LIN {X -174.485,Y -231.635,Z 231.220,A 53.010,B 90.000,C 0.000} C_DIS
LIN {X -172.527,Y -233.097,Z 231.745,A 53.493,B 90.000,C 0.000} C_DIS
LIN {X -170.564,Y -234.537,Z 232.313,A 53.974,B 90.000,C 0.000} C_DIS
LIN {X -168.598,Y -235.954,Z 232.925,A 54.453,B 90.000,C 0.000} C_DIS
LIN {X -166.629,Y -237.349,Z 233.579,A 54.929,B 90.000,C 0.000} C_DIS
LIN {X -164.658,Y -238.720,Z 234.275,A 55.404,B 90.000,C 0.000} C_DIS
LIN {X -162.687,Y -240.067,Z 235.015,A 55.876,B 90.000,C 0.000} C_DIS
LIN {X -160.716,Y -241.392,Z 235.795,A 56.345,B 90.000,C 0.000} C_DIS
LIN {X -158.746,Y -242.692,Z 236.618,A 56.811,B 90.000,C 0.000} C_DIS
LIN {X -157.556,Y -243.467,Z 237.135,A 57.092,B 90.000,C 0.000} C_DIS
LIN {X -156.469,Y -241.788,Z 237.135,A 57.092,B 90.000,C 0.000} C_DIS
WAIT SEC 0.1
RET=EKI_SetBool("oxy","torchState",FALSE)
RET = EKI_Send("oxy","torchState")
LIN {X -146.690,Y -226.676,Z 237.135,A 57.092,B 90.000,C 0.000} C_DIS
LIN {X -123.076,Y -240.317,Z 224.158,A 62.881,B 90.000,C 0.000} C_DIS
LIN {X -131.281,Y -256.338,Z 224.158,A 62.881,B 90.000,C 0.000} C_DIS
LIN {X -132.192,Y -258.119,Z 224.158,A 62.881,B 90.000,C 0.000} C_DIS
WAIT SEC 1.75
RET=EKI_SetBool("oxy","torchState",TRUE)
RET = EKI_Send("oxy","torchState")
LIN {X -129.997,Y -259.231,Z 224.597,A 63.368,B 90.000,C 0.000} C_DIS
LIN {X -127.784,Y -260.329,Z 224.980,A 63.856,B 90.000,C 0.000} C_DIS
LIN {X -125.556,Y -261.409,Z 225.324,A 64.345,B 90.000,C 0.000} C_DIS
LIN {X -123.317,Y -262.472,Z 225.647,A 64.834,B 90.000,C 0.000} C_DIS
LIN {X -121.069,Y -263.517,Z 225.964,A 65.324,B 90.000,C 0.000} C_DIS
LIN {X -118.813,Y -264.544,Z 226.289,A 65.814,B 90.000,C 0.000} C_DIS
LIN {X -116.551,Y -265.548,Z 226.642,A 66.303,B 90.000,C 0.000} C_DIS
LIN {X -114.287,Y -266.530,Z 227.038,A 66.791,B 90.000,C 0.000} C_DIS
LIN {X -112.023,Y -267.490,Z 227.491,A 67.276,B 90.000,C 0.000} C_DIS
LIN {X -109.763,Y -268.425,Z 228.003,A 67.760,B 90.000,C 0.000} C_DIS
LIN {X -107.506,Y -269.337,Z 228.573,A 68.241,B 90.000,C 0.000} C_DIS
LIN {X -105.255,Y -270.224,Z 229.202,A 68.719,B 90.000,C 0.000} C_DIS
LIN {X -103.012,Y -271.087,Z 229.888,A 69.193,B 90.000,C 0.000} C_DIS
LIN {X -100.777,Y -271.926,Z 230.630,A 69.665,B 90.000,C 0.000} C_DIS
LIN {X -98.553,Y -272.740,Z 231.430,A 70.133,B 90.000,C 0.000} C_DIS
LIN {X -96.341,Y -273.529,Z 232.285,A 70.597,B 90.000,C 0.000} C_DIS
LIN {X -94.142,Y -274.293,Z 233.197,A 71.057,B 90.000,C 0.000} C_DIS
LIN {X -91.959,Y -275.033,Z 234.163,A 71.512,B 90.000,C 0.000} C_DIS
LIN {X -89.792,Y -275.748,Z 235.184,A 71.963,B 90.000,C 0.000} C_DIS
LIN {X -87.644,Y -276.439,Z 236.259,A 72.409,B 90.000,C 0.000} C_DIS
LIN {X -85.515,Y -277.105,Z 237.388,A 72.850,B 90.000,C 0.000} C_DIS
LIN {X -85.176,Y -277.209,Z 237.573,A 72.920,B 90.000,C 0.000} C_DIS
LIN {X -84.588,Y -275.298,Z 237.573,A 72.920,B 90.000,C 0.000} C_DIS
WAIT SEC 0.1
RET=EKI_SetBool("oxy","torchState",FALSE)
RET = EKI_Send("oxy","torchState")
LIN {X -79.302,Y -258.092,Z 237.573,A 72.920,B 90.000,C 0.000} C_DIS
LIN {X -88.721,Y -255.007,Z 203.676,A 70.816,B 90.000,C 0.000} C_DIS
LIN {X -94.636,Y -272.007,Z 203.676,A 70.816,B 90.000,C 0.000} C_DIS
LIN {X -95.293,Y -273.896,Z 203.676,A 70.816,B 90.000,C 0.000} C_DIS
WAIT SEC 1.75
RET=EKI_SetBool("oxy","torchState",TRUE)
RET = EKI_Send("oxy","torchState")
LIN {X -97.616,Y -273.077,Z 203.247,A 70.330,B 90.000,C 0.000} C_DIS
LIN {X -99.938,Y -272.235,Z 202.861,A 69.842,B 90.000,C 0.000} C_DIS
LIN {X -102.254,Y -271.373,Z 202.486,A 69.354,B 90.000,C 0.000} C_DIS
LIN {X -104.561,Y -270.494,Z 202.097,A 68.866,B 90.000,C 0.000} C_DIS
LIN {X -106.853,Y -269.596,Z 201.662,A 68.379,B 90.000,C 0.000} C_DIS
LIN {X -109.130,Y -268.682,Z 201.183,A 67.895,B 90.000,C 0.000} C_DIS
LIN {X -111.390,Y -267.754,Z 200.657,A 67.412,B 90.000,C 0.000} C_DIS
LIN {X -113.632,Y -266.810,Z 200.082,A 66.931,B 90.000,C 0.000} C_DIS
LIN {X -115.856,Y -265.851,Z 199.461,A 66.453,B 90.000,C 0.000} C_DIS
LIN {X -118.061,Y -264.880,Z 198.796,A 65.977,B 90.000,C 0.000} C_DIS
LIN {X -120.246,Y -263.896,Z 198.084,A 65.503,B 90.000,C 0.000} C_DIS
LIN {X -122.409,Y -262.899,Z 197.325,A 65.033,B 90.000,C 0.000} C_DIS
LIN {X -124.550,Y -261.891,Z 196.521,A 64.565,B 90.000,C 0.000} C_DIS
LIN {X -126.670,Y -260.873,Z 195.673,A 64.101,B 90.000,C 0.000} C_DIS
LIN {X -128.766,Y -259.845,Z 194.779,A 63.639,B 90.000,C 0.000} C_DIS
LIN {X -130.837,Y -258.807,Z 193.840,A 63.182,B 90.000,C 0.000} C_DIS
LIN {X -132.884,Y -257.762,Z 192.856,A 62.728,B 90.000,C 0.000} C_DIS
LIN {X -134.776,Y -256.779,Z 191.899,A 62.306,B 90.000,C 0.000} C_DIS
LIN {X -133.846,Y -255.008,Z 191.899,A 62.306,B 90.000,C 0.000} C_DIS
WAIT SEC 0.1
RET=EKI_SetBool("oxy","torchState",FALSE)
RET = EKI_Send("oxy","torchState")
LIN {X -125.481,Y -239.070,Z 191.899,A 62.306,B 90.000,C 0.000} C_DIS
LIN {X -100.690,Y -250.523,Z 169.381,A 68.104,B 90.000,C 0.000} C_DIS
LIN {X -107.403,Y -267.224,Z 169.381,A 68.104,B 90.000,C 0.000} C_DIS
LIN {X -108.148,Y -269.080,Z 169.381,A 68.104,B 90.000,C 0.000} C_DIS
WAIT SEC 1.75
RET=EKI_SetBool("oxy","torchState",TRUE)
RET = EKI_Send("oxy","torchState")
LIN {X -105.841,Y -269.995,Z 169.670,A 68.594,B 90.000,C 0.000} C_DIS
LIN {X -103.520,Y -270.893,Z 169.913,A 69.086,B 90.000,C 0.000} C_DIS
LIN {X -101.192,Y -271.772,Z 170.145,A 69.578,B 90.000,C 0.000} C_DIS
LIN {X -98.858,Y -272.630,Z 170.404,A 70.069,B 90.000,C 0.000} C_DIS
LIN {X -96.524,Y -273.464,Z 170.725,A 70.559,B 90.000,C 0.000} C_DIS
LIN {X -94.192,Y -274.276,Z 171.117,A 71.046,B 90.000,C 0.000} C_DIS
LIN {X -91.865,Y -275.065,Z 171.577,A 71.532,B 90.000,C 0.000} C_DIS
LIN {X -89.544,Y -275.829,Z 172.102,A 72.015,B 90.000,C 0.000} C_DIS
LIN {X -87.230,Y -276.569,Z 172.690,A 72.495,B 90.000,C 0.000} C_DIS
LIN {X -84.924,Y -277.286,Z 173.335,A 72.972,B 90.000,C 0.000} C_DIS
LIN {X -82.626,Y -277.979,Z 174.034,A 73.446,B 90.000,C 0.000} C_DIS
LIN {X -80.337,Y -278.649,Z 174.783,A 73.917,B 90.000,C 0.000} C_DIS
LIN {X -78.058,Y -279.297,Z 175.578,A 74.385,B 90.000,C 0.000} C_DIS
LIN {X -75.788,Y -279.921,Z 176.419,A 74.851,B 90.000,C 0.000} C_DIS
LIN {X -73.526,Y -280.523,Z 177.298,A 75.313,B 90.000,C 0.000} C_DIS
LIN {X -71.273,Y -281.105,Z 178.212,A 75.773,B 90.000,C 0.000} C_DIS
LIN {X -69.029,Y -281.664,Z 179.160,A 76.230,B 90.000,C 0.000} C_DIS
LIN {X -66.792,Y -282.203,Z 180.136,A 76.684,B 90.000,C 0.000} C_DIS
LIN {X -64.561,Y -282.722,Z 181.137,A 77.137,B 90.000,C 0.000} C_DIS
LIN {X -62.337,Y -283.220,Z 182.163,A 77.587,B 90.000,C 0.000} C_DIS
LIN {X -60.117,Y -283.699,Z 183.208,A 78.036,B 90.000,C 0.000} C_DIS
LIN {X -57.901,Y -284.159,Z 184.270,A 78.483,B 90.000,C 0.000} C_DIS
LIN {X -55.688,Y -284.600,Z 185.345,A 78.929,B 90.000,C 0.000} C_DIS
LIN {X -53.477,Y -285.024,Z 186.431,A 79.374,B 90.000,C 0.000} C_DIS
LIN {X -51.266,Y -285.431,Z 187.524,A 79.818,B 90.000,C 0.000} C_DIS
LIN {X -49.054,Y -285.816,Z 188.623,A 80.261,B 90.000,C 0.000} C_DIS
LIN {X -47.559,Y -286.074,Z 189.367,A 80.561,B 90.000,C 0.000} C_DIS
LIN {X -47.231,Y -284.101,Z 189.367,A 80.561,B 90.000,C 0.000} C_DIS
WAIT SEC 0.1
RET=EKI_SetBool("oxy","torchState",FALSE)
RET = EKI_Send("oxy","torchState")
LIN {X -44.279,Y -266.344,Z 189.367,A 80.561,B 90.000,C 0.000} C_DIS
LIN {X -23.730,Y -268.955,Z 178.464,A 84.958,B 90.000,C 0.000} C_DIS
LIN {X -25.312,Y -286.885,Z 178.464,A 84.958,B 90.000,C 0.000} C_DIS
LIN {X -25.488,Y -288.878,Z 178.464,A 84.958,B 90.000,C 0.000} C_DIS
WAIT SEC 1.75
RET=EKI_SetBool("oxy","torchState",TRUE)
RET = EKI_Send("oxy","torchState")
LIN {X -27.825,Y -288.662,Z 177.602,A 84.494,B 90.000,C 0.000} C_DIS
LIN {X -30.135,Y -288.429,Z 176.676,A 84.035,B 90.000,C 0.000} C_DIS
LIN {X -32.420,Y -288.182,Z 175.693,A 83.581,B 90.000,C 0.000} C_DIS
LIN {X -34.681,Y -287.919,Z 174.660,A 83.132,B 90.000,C 0.000} C_DIS
LIN {X -36.919,Y -287.640,Z 173.581,A 82.686,B 90.000,C 0.000} C_DIS
LIN {X -39.139,Y -287.347,Z 172.471,A 82.244,B 90.000,C 0.000} C_DIS
LIN {X -41.342,Y -287.038,Z 171.331,A 81.804,B 90.000,C 0.000} C_DIS
LIN {X -43.532,Y -286.713,Z 170.171,A 81.367,B 90.000,C 0.000} C_DIS
LIN {X -45.713,Y -286.374,Z 168.998,A 80.931,B 90.000,C 0.000} C_DIS
LIN {X -47.888,Y -286.018,Z 167.817,A 80.495,B 90.000,C 0.000} C_DIS
LIN {X -50.060,Y -285.644,Z 166.638,A 80.060,B 90.000,C 0.000} C_DIS
LIN {X -52.233,Y -285.256,Z 165.466,A 79.624,B 90.000,C 0.000} C_DIS
LIN {X -54.410,Y -284.849,Z 164.306,A 79.186,B 90.000,C 0.000} C_DIS
LIN {X -56.595,Y -284.423,Z 163.169,A 78.746,B 90.000,C 0.000} C_DIS
LIN {X -58.790,Y -283.978,Z 162.059,A 78.304,B 90.000,C 0.000} C_DIS
LIN {X -60.381,Y -283.644,Z 161.280,A 77.983,B 90.000,C 0.000} C_DIS
LIN {X -59.964,Y -281.688,Z 161.280,A 77.983,B 90.000,C 0.000} C_DIS
WAIT SEC 0.1
RET=EKI_SetBool("oxy","torchState",FALSE)
RET = EKI_Send("oxy","torchState")
LIN {X -56.216,Y -264.083,Z 161.280,A 77.983,B 90.000,C 0.000} C_DIS
LIN {X -40.841,Y -266.893,Z 146.065,A 81.300,B 90.000,C 0.000} C_DIS
LIN {X -43.563,Y -284.686,Z 146.065,A 81.300,B 90.000,C 0.000} C_DIS
LIN {X -43.866,Y -286.663,Z 146.065,A 81.300,B 90.000,C 0.000} C_DIS
WAIT SEC 1.75
RET=EKI_SetBool("oxy","torchState",TRUE)
RET = EKI_Send("oxy","torchState")
LIN {X -41.493,Y -287.012,Z 146.771,A 81.774,B 90.000,C 0.000} C_DIS
LIN {X -39.121,Y -287.344,Z 147.484,A 82.247,B 90.000,C 0.000} C_DIS
LIN {X -36.747,Y -287.661,Z 148.202,A 82.720,B 90.000,C 0.000} C_DIS
LIN {X -34.373,Y -287.952,Z 148.929,A 83.193,B 90.000,C 0.000} C_DIS
LIN {X -32.000,Y -288.224,Z 149.663,A 83.665,B 90.000,C 0.000} C_DIS
LIN {X -29.626,Y -288.481,Z 150.403,A 84.137,B 90.000,C 0.000} C_DIS
LIN {X -27.252,Y -288.713,Z 151.151,A 84.608,B 90.000,C 0.000} C_DIS
LIN {X -24.879,Y -288.926,Z 151.907,A 85.079,B 90.000,C 0.000} C_DIS
LIN {X -22.506,Y -289.123,Z 152.668,A 85.549,B 90.000,C 0.000} C_DIS
LIN {X -20.134,Y -289.297,Z 153.437,A 86.019,B 90.000,C 0.000} C_DIS
LIN {X -18.908,Y -289.383,Z 153.837,A 86.262,B 90.000,C 0.000} C_DIS
LIN {X -18.777,Y -287.387,Z 153.837,A 86.262,B 90.000,C 0.000} C_DIS
WAIT SEC 0.1
RET=EKI_SetBool("oxy","torchState",FALSE)
RET = EKI_Send("oxy","torchState")
LIN {X -17.604,Y -269.426,Z 153.837,A 86.262,B 90.000,C 0.000} C_DIS
LIN {X 5.612,Y -269.942,Z 139.862,A 91.191,B 90.000,C 0.000} C_DIS
LIN {X 5.986,Y -287.938,Z 139.862,A 91.191,B 90.000,C 0.000} C_DIS
LIN {X 6.028,Y -289.937,Z 139.862,A 91.191,B 90.000,C 0.000} C_DIS
WAIT SEC 1.75
RET=EKI_SetBool("oxy","torchState",TRUE)
RET = EKI_Send("oxy","torchState")
LIN {X 8.397,Y -289.878,Z 140.657,A 91.659,B 90.000,C 0.000} C_DIS
LIN {X 10.728,Y -289.801,Z 141.555,A 92.120,B 90.000,C 0.000} C_DIS
LIN {X 13.001,Y -289.708,Z 142.592,A 92.569,B 90.000,C 0.000} C_DIS
LIN {X 15.183,Y -289.602,Z 143.807,A 93.001,B 90.000,C 0.000} C_DIS
LIN {X 17.238,Y -289.487,Z 145.226,A 93.408,B 90.000,C 0.000} C_DIS
LIN {X 19.120,Y -289.369,Z 146.866,A 93.780,B 90.000,C 0.000} C_DIS
LIN {X 20.776,Y -289.255,Z 148.735,A 94.108,B 90.000,C 0.000} C_DIS
LIN {X 22.142,Y -289.153,Z 150.827,A 94.379,B 90.000,C 0.000} C_DIS
LIN {X 22.275,Y -289.143,Z 151.073,A 94.405,B 90.000,C 0.000} C_DIS
LIN {X 22.122,Y -287.149,Z 151.073,A 94.405,B 90.000,C 0.000} C_DIS
WAIT SEC 0.1
RET=EKI_SetBool("oxy","torchState",FALSE)
RET = EKI_Send("oxy","torchState")
LIN {X 20.739,Y -269.202,Z 151.073,A 94.405,B 90.000,C 0.000} C_DIS
LIN {X 20.977,Y -269.184,Z 165.846,A 94.456,B 90.000,C 0.000} C_DIS
LIN {X 22.376,Y -287.129,Z 165.846,A 94.456,B 90.000,C 0.000} C_DIS
LIN {X 22.531,Y -289.123,Z 165.846,A 94.456,B 90.000,C 0.000} C_DIS
WAIT SEC 1.75
RET=EKI_SetBool("oxy","torchState",TRUE)
RET = EKI_Send("oxy","torchState")
LIN {X 21.416,Y -289.208,Z 168.082,A 94.235,B 90.000,C 0.000} C_DIS
LIN {X 20.047,Y -289.306,Z 170.171,A 93.964,B 90.000,C 0.000} C_DIS
LIN {X 18.459,Y -289.412,Z 172.099,A 93.649,B 90.000,C 0.000} C_DIS
LIN {X 16.685,Y -289.520,Z 173.857,A 93.298,B 90.000,C 0.000} C_DIS
LIN {X 14.754,Y -289.624,Z 175.441,A 92.916,B 90.000,C 0.000} C_DIS
LIN {X 12.689,Y -289.722,Z 176.845,A 92.508,B 90.000,C 0.000} C_DIS
LIN {X 10.513,Y -289.809,Z 178.073,A 92.078,B 90.000,C 0.000} C_DIS
LIN {X 8.247,Y -289.883,Z 179.127,A 91.630,B 90.000,C 0.000} C_DIS
LIN {X 5.908,Y -289.940,Z 180.005,A 91.167,B 90.000,C 0.000} C_DIS
LIN {X 3.512,Y -289.979,Z 180.716,A 90.694,B 90.000,C 0.000} C_DIS
LIN {X 1.073,Y -289.998,Z 181.264,A 90.212,B 90.000,C 0.000} C_DIS
LIN {X -1.396,Y -289.997,Z 181.653,A 89.724,B 90.000,C 0.000} C_DIS
LIN {X -3.885,Y -289.974,Z 181.888,A 89.232,B 90.000,C 0.000} C_DIS
LIN {X -6.286,Y -289.932,Z 181.974,A 88.758,B 90.000,C 0.000} C_DIS
LIN {X -6.243,Y -287.932,Z 181.974,A 88.758,B 90.000,C 0.000} C_DIS
WAIT SEC 0.1
RET=EKI_SetBool("oxy","torchState",FALSE)
RET = EKI_Send("oxy","torchState")
LIN {X -5.852,Y -269.937,Z 181.974,A 88.758,B 90.000,C 0.000} C_DIS
LIN {X -12.189,Y -269.725,Z 203.494,A 87.412,B 90.000,C 0.000} C_DIS
LIN {X -13.002,Y -287.706,Z 203.494,A 87.412,B 90.000,C 0.000} C_DIS
LIN {X -13.092,Y -289.704,Z 203.494,A 87.412,B 90.000,C 0.000} C_DIS
WAIT SEC 1.75
RET=EKI_SetBool("oxy","torchState",TRUE)
RET = EKI_Send("oxy","torchState")
LIN {X -10.663,Y -289.804,Z 204.075,A 87.893,B 90.000,C 0.000} C_DIS
LIN {X -8.217,Y -289.883,Z 204.584,A 88.376,B 90.000,C 0.000} C_DIS
LIN {X -5.755,Y -289.942,Z 205.016,A 88.863,B 90.000,C 0.000} C_DIS
LIN {X -3.281,Y -289.981,Z 205.369,A 89.352,B 90.000,C 0.000} C_DIS
LIN {X -0.796,Y -289.999,Z 205.637,A 89.843,B 90.000,C 0.000} C_DIS
LIN {X 1.698,Y -289.995,Z 205.815,A 90.335,B 90.000,C 0.000} C_DIS
LIN {X 4.196,Y -289.970,Z 205.903,A 90.829,B 90.000,C 0.000} C_DIS
LIN {X 6.695,Y -289.922,Z 205.890,A 91.323,B 90.000,C 0.000} C_DIS
LIN {X 9.191,Y -289.854,Z 205.779,A 91.816,B 90.000,C 0.000} C_DIS
LIN {X 11.679,Y -289.764,Z 205.556,A 92.308,B 90.000,C 0.000} C_DIS
LIN {X 14.154,Y -289.654,Z 205.224,A 92.798,B 90.000,C 0.000} C_DIS
LIN {X 16.610,Y -289.524,Z 204.776,A 93.283,B 90.000,C 0.000} C_DIS
LIN {X 19.039,Y -289.374,Z 204.206,A 93.764,B 90.000,C 0.000} C_DIS
LIN {X 21.435,Y -289.206,Z 203.512,A 94.239,B 90.000,C 0.000} C_DIS
LIN {X 23.790,Y -289.023,Z 202.694,A 94.705,B 90.000,C 0.000} C_DIS
LIN {X 23.626,Y -287.029,Z 202.694,A 94.705,B 90.000,C 0.000} C_DIS
WAIT SEC 0.1
RET=EKI_SetBool("oxy","torchState",FALSE)
RET = EKI_Send("oxy","torchState")
LIN {X 22.149,Y -269.090,Z 202.694,A 94.705,B 90.000,C 0.000} C_DIS
LIN {X 39.945,Y -267.029,Z 190.477,A 98.508,B 90.000,C 0.000} C_DIS
LIN {X 42.608,Y -284.831,Z 190.477,A 98.508,B 90.000,C 0.000} C_DIS
LIN {X 42.904,Y -286.809,Z 190.477,A 98.508,B 90.000,C 0.000} C_DIS
WAIT SEC 1.75
RET=EKI_SetBool("oxy","torchState",TRUE)
RET = EKI_Send("oxy","torchState")
LIN {X 44.729,Y -286.530,Z 188.792,A 98.873,B 90.000,C 0.000} C_DIS
LIN {X 46.502,Y -286.247,Z 187.053,A 99.227,B 90.000,C 0.000} C_DIS
LIN {X 48.216,Y -285.963,Z 185.256,A 99.571,B 90.000,C 0.000} C_DIS
LIN {X 49.864,Y -285.681,Z 183.398,A 99.901,B 90.000,C 0.000} C_DIS
LIN {X 51.432,Y -285.403,Z 181.471,A 100.216,B 90.000,C 0.000} C_DIS
LIN {X 52.915,Y -285.131,Z 179.477,A 100.513,B 90.000,C 0.000} C_DIS
LIN {X 54.300,Y -284.871,Z 177.412,A 100.792,B 90.000,C 0.000} C_DIS
LIN {X 55.573,Y -284.625,Z 175.275,A 101.048,B 90.000,C 0.000} C_DIS
LIN {X 56.724,Y -284.398,Z 173.068,A 101.280,B 90.000,C 0.000} C_DIS
LIN {X 57.368,Y -284.269,Z 171.672,A 101.410,B 90.000,C 0.000} C_DIS
LIN {X 56.973,Y -282.309,Z 171.672,A 101.410,B 90.000,C 0.000} C_DIS
WAIT SEC 0.1
RET=EKI_SetBool("oxy","torchState",FALSE)
RET = EKI_Send("oxy","torchState")
LIN {X 53.412,Y -264.664,Z 171.672,A 101.410,B 90.000,C 0.000} C_DIS
LIN {X 54.636,Y -264.414,Z 148.285,A 101.675,B 90.000,C 0.000} C_DIS
LIN {X 58.279,Y -282.042,Z 148.285,A 101.675,B 90.000,C 0.000} C_DIS
LIN {X 58.684,Y -284.000,Z 148.285,A 101.675,B 90.000,C 0.000} C_DIS
WAIT SEC 1.75
RET=EKI_SetBool("oxy","torchState",TRUE)
RET = EKI_Send("oxy","torchState")
LIN {X 57.692,Y -284.204,Z 146.000,A 101.475,B 90.000,C 0.000} C_DIS
LIN {X 56.490,Y -284.445,Z 143.821,A 101.233,B 90.000,C 0.000} C_DIS
LIN {X 55.104,Y -284.717,Z 141.759,A 100.954,B 90.000,C 0.000} C_DIS
LIN {X 53.557,Y -285.012,Z 139.817,A 100.642,B 90.000,C 0.000} C_DIS
LIN {X 51.869,Y -285.324,Z 138.000,A 100.303,B 90.000,C 0.000} C_DIS
LIN {X 50.060,Y -285.646,Z 136.306,A 99.940,B 90.000,C 0.000} C_DIS
LIN {X 48.146,Y -285.975,Z 134.731,A 99.557,B 90.000,C 0.000} C_DIS
LIN {X 47.860,Y -286.023,Z 134.510,A 99.499,B 90.000,C 0.000} C_DIS
LIN {X 47.530,Y -284.051,Z 134.510,A 99.499,B 90.000,C 0.000} C_DIS
WAIT SEC 0.1
RET=EKI_SetBool("oxy","torchState",FALSE)
RET = EKI_Send("oxy","torchState")
LIN {X 44.559,Y -266.298,Z 134.510,A 99.499,B 90.000,C 0.000} C_DIS
LIN {X 30.080,Y -268.319,Z 126.079,A 96.396,B 90.000,C 0.000} C_DIS
LIN {X 32.085,Y -286.207,Z 126.079,A 96.396,B 90.000,C 0.000} C_DIS
LIN {X 32.308,Y -288.195,Z 126.079,A 96.396,B 90.000,C 0.000} C_DIS
WAIT SEC 1.75
RET=EKI_SetBool("oxy","torchState",TRUE)
RET = EKI_Send("oxy","torchState")
LIN {X 30.008,Y -288.442,Z 125.131,A 95.939,B 90.000,C 0.000} C_DIS
LIN {X 27.696,Y -288.674,Z 124.211,A 95.480,B 90.000,C 0.000} C_DIS
LIN {X 25.369,Y -288.887,Z 123.323,A 95.019,B 90.000,C 0.000} C_DIS
LIN {X 23.028,Y -289.083,Z 122.466,A 94.555,B 90.000,C 0.000} C_DIS
LIN {X 20.675,Y -289.261,Z 121.643,A 94.088,B 90.000,C 0.000} C_DIS
LIN {X 18.308,Y -289.421,Z 120.853,A 93.620,B 90.000,C 0.000} C_DIS
LIN {X 15.929,Y -289.561,Z 120.099,A 93.149,B 90.000,C 0.000} C_DIS
LIN {X 13.538,Y -289.683,Z 119.381,A 92.676,B 90.000,C 0.000} C_DIS
LIN {X 11.135,Y -289.785,Z 118.702,A 92.200,B 90.000,C 0.000} C_DIS
LIN {X 8.720,Y -289.869,Z 118.059,A 91.723,B 90.000,C 0.000} C_DIS
LIN {X 6.295,Y -289.931,Z 117.459,A 91.244,B 90.000,C 0.000} C_DIS
LIN {X 3.859,Y -289.974,Z 116.898,A 90.762,B 90.000,C 0.000} C_DIS
LIN {X 1.414,Y -289.996,Z 116.380,A 90.279,B 90.000,C 0.000} C_DIS
LIN {X -1.041,Y -289.997,Z 115.907,A 89.794,B 90.000,C 0.000} C_DIS
LIN {X -3.503,Y -289.978,Z 115.477,A 89.308,B 90.000,C 0.000} C_DIS
LIN {X -5.973,Y -289.938,Z 115.094,A 88.820,B 90.000,C 0.000} C_DIS
LIN {X -8.450,Y -289.876,Z 114.760,A 88.330,B 90.000,C 0.000} C_DIS
LIN {X -10.931,Y -289.793,Z 114.474,A 87.840,B 90.000,C 0.000} C_DIS
LIN {X -13.418,Y -289.689,Z 114.237,A 87.348,B 90.000,C 0.000} C_DIS
LIN {X -15.907,Y -289.563,Z 114.051,A 86.856,B 90.000,C 0.000} C_DIS
LIN {X -18.399,Y -289.415,Z 113.920,A 86.362,B 90.000,C 0.000} C_DIS
LIN {X -20.892,Y -289.246,Z 113.843,A 85.869,B 90.000,C 0.000} C_DIS
LIN {X -23.384,Y -289.055,Z 113.821,A 85.375,B 90.000,C 0.000} C_DIS
LIN {X -25.875,Y -288.843,Z 113.854,A 84.881,B 90.000,C 0.000} C_DIS
LIN {X -26.365,Y -288.799,Z 113.866,A 84.784,B 90.000,C 0.000} C_DIS
LIN {X -26.184,Y -286.807,Z 113.866,A 84.784,B 90.000,C 0.000} C_DIS
WAIT SEC 0.1
RET=EKI_SetBool("oxy","torchState",FALSE)
RET = EKI_Send("oxy","torchState")
LIN {X -24.547,Y -268.882,Z 113.866,A 84.784,B 90.000,C 0.000} C_DIS
LIN {X -36.877,Y -267.470,Z 113.990,A 82.150,B 90.000,C 0.000} C_DIS
LIN {X -39.336,Y -285.301,Z 113.990,A 82.150,B 90.000,C 0.000} C_DIS
LIN {X -39.609,Y -287.282,Z 113.990,A 82.150,B 90.000,C 0.000} C_DIS
WAIT SEC 1.75
RET=EKI_SetBool("oxy","torchState",TRUE)
RET = EKI_Send("oxy","torchState")
LIN {X -42.062,Y -286.933,Z 113.662,A 81.660,B 90.000,C 0.000} C_DIS
LIN {X -44.477,Y -286.569,Z 113.127,A 81.178,B 90.000,C 0.000} C_DIS
LIN {X -46.822,Y -286.195,Z 112.348,A 80.709,B 90.000,C 0.000} C_DIS
LIN {X -49.059,Y -285.820,Z 111.296,A 80.261,B 90.000,C 0.000} C_DIS
LIN {X -51.128,Y -285.457,Z 109.942,A 79.845,B 90.000,C 0.000} C_DIS
LIN {X -52.966,Y -285.122,Z 108.282,A 79.476,B 90.000,C 0.000} C_DIS
LIN {X -54.526,Y -284.828,Z 106.351,A 79.163,B 90.000,C 0.000} C_DIS
LIN {X -55.790,Y -284.583,Z 104.208,A 78.908,B 90.000,C 0.000} C_DIS
LIN {X -56.744,Y -284.394,Z 101.905,A 78.716,B 90.000,C 0.000} C_DIS
LIN {X -57.169,Y -284.309,Z 100.461,A 78.631,B 90.000,C 0.000} C_DIS
LIN {X -56.774,Y -282.348,Z 100.461,A 78.631,B 90.000,C 0.000} C_DIS
WAIT SEC 0.1
RET=EKI_SetBool("oxy","torchState",FALSE)
RET = EKI_Send("oxy","torchState")
LIN {X -53.226,Y -264.702,Z 100.461,A 78.631,B 90.000,C 0.000} C_DIS
LIN {X -60.163,Y -263.212,Z 120.264,A 77.125,B 90.000,C 0.000} C_DIS
LIN {X -64.173,Y -280.759,Z 120.264,A 77.125,B 90.000,C 0.000} C_DIS
LIN {X -64.619,Y -282.709,Z 120.264,A 77.125,B 90.000,C 0.000} C_DIS
WAIT SEC 1.75
RET=EKI_SetBool("oxy","torchState",TRUE)
RET = EKI_Send("oxy","torchState")
LIN {X -62.571,Y -283.169,Z 121.622,A 77.540,B 90.000,C 0.000} C_DIS
LIN {X -60.462,Y -283.627,Z 122.883,A 77.966,B 90.000,C 0.000} C_DIS
LIN {X -58.301,Y -284.079,Z 124.056,A 78.402,B 90.000,C 0.000} C_DIS
LIN {X -56.093,Y -284.523,Z 125.139,A 78.847,B 90.000,C 0.000} C_DIS
LIN {X -53.844,Y -284.957,Z 126.141,A 79.300,B 90.000,C 0.000} C_DIS
LIN {X -51.560,Y -285.380,Z 127.064,A 79.759,B 90.000,C 0.000} C_DIS
LIN {X -49.244,Y -285.788,Z 127.912,A 80.223,B 90.000,C 0.000} C_DIS
LIN {X -46.902,Y -286.182,Z 128.691,A 80.693,B 90.000,C 0.000} C_DIS
LIN {X -44.537,Y -286.559,Z 129.408,A 81.166,B 90.000,C 0.000} C_DIS
LIN {X -42.359,Y -286.890,Z 130.012,A 81.601,B 90.000,C 0.000} C_DIS
LIN {X -42.067,Y -284.911,Z 130.012,A 81.601,B 90.000,C 0.000} C_DIS
WAIT SEC 0.1
RET=EKI_SetBool("oxy","torchState",FALSE)
RET = EKI_Send("oxy","torchState")
LIN {X -39.438,Y -267.104,Z 130.012,A 81.601,B 90.000,C 0.000} C_DIS
LIN {X -74.388,Y -259.551,Z 101.612,A 74.008,B 90.000,C 0.000} C_DIS
LIN {X -79.347,Y -276.854,Z 101.612,A 74.008,B 90.000,C 0.000} C_DIS
LIN {X -79.898,Y -278.777,Z 101.612,A 74.008,B 90.000,C 0.000} C_DIS
WAIT SEC 1.75
RET=EKI_SetBool("oxy","torchState",TRUE)
RET = EKI_Send("oxy","torchState")
LIN {X -80.728,Y -278.537,Z 99.266,A 73.837,B 90.000,C 0.000} C_DIS
LIN {X -81.396,Y -278.343,Z 96.865,A 73.699,B 90.000,C 0.000} C_DIS
LIN {X -81.903,Y -278.194,Z 94.422,A 73.595,B 90.000,C 0.000} C_DIS
LIN {X -82.243,Y -278.094,Z 91.947,A 73.525,B 90.000,C 0.000} C_DIS
LIN {X -82.420,Y -278.041,Z 89.454,A 73.488,B 90.000,C 0.000} C_DIS
LIN {X -82.435,Y -278.037,Z 86.955,A 73.485,B 90.000,C 0.000} C_DIS
LIN {X -82.285,Y -278.081,Z 84.460,A 73.516,B 90.000,C 0.000} C_DIS
LIN {X -81.969,Y -278.175,Z 81.982,A 73.582,B 90.000,C 0.000} C_DIS
LIN {X -81.493,Y -278.314,Z 79.532,A 73.679,B 90.000,C 0.000} C_DIS
LIN {X -80.862,Y -278.498,Z 77.120,A 73.809,B 90.000,C 0.000} C_DIS
LIN {X -80.077,Y -278.725,Z 74.758,A 73.971,B 90.000,C 0.000} C_DIS
LIN {X -79.144,Y -278.991,Z 72.454,A 74.162,B 90.000,C 0.000} C_DIS
LIN {X -78.069,Y -279.294,Z 70.218,A 74.383,B 90.000,C 0.000} C_DIS
LIN {X -76.855,Y -279.631,Z 68.059,A 74.632,B 90.000,C 0.000} C_DIS
LIN {X -76.252,Y -279.796,Z 67.095,A 74.755,B 90.000,C 0.000} C_DIS
LIN {X -75.726,Y -277.866,Z 67.095,A 74.755,B 90.000,C 0.000} C_DIS
WAIT SEC 0.1
RET=EKI_SetBool("oxy","torchState",FALSE)
RET = EKI_Send("oxy","torchState")
LIN {X -70.994,Y -260.499,Z 67.095,A 74.755,B 90.000,C 0.000} C_DIS
LIN {X -71.477,Y -260.367,Z 43.916,A 74.649,B 90.000,C 0.000} C_DIS
LIN {X -76.242,Y -277.725,Z 43.916,A 74.649,B 90.000,C 0.000} C_DIS
LIN {X -76.772,Y -279.654,Z 43.916,A 74.649,B 90.000,C 0.000} C_DIS
WAIT SEC 1.75
RET=EKI_SetBool("oxy","torchState",TRUE)
RET = EKI_Send("oxy","torchState")
LIN {X -79.027,Y -279.023,Z 44.789,A 74.186,B 90.000,C 0.000} C_DIS
LIN {X -81.275,Y -278.378,Z 45.673,A 73.724,B 90.000,C 0.000} C_DIS
LIN {X -83.506,Y -277.717,Z 46.585,A 73.265,B 90.000,C 0.000} C_DIS
LIN {X -85.712,Y -277.044,Z 47.550,A 72.809,B 90.000,C 0.000} C_DIS
LIN {X -87.883,Y -276.363,Z 48.585,A 72.359,B 90.000,C 0.000} C_DIS
LIN {X -90.009,Y -275.678,Z 49.708,A 71.918,B 90.000,C 0.000} C_DIS
LIN {X -92.072,Y -274.996,Z 50.943,A 71.489,B 90.000,C 0.000} C_DIS
LIN {X -94.061,Y -274.322,Z 52.298,A 71.074,B 90.000,C 0.000} C_DIS
LIN {X -95.956,Y -273.665,Z 53.791,A 70.678,B 90.000,C 0.000} C_DIS
LIN {X -97.736,Y -273.034,Z 55.428,A 70.304,B 90.000,C 0.000} C_DIS
LIN {X -99.376,Y -272.441,Z 57.219,A 69.960,B 90.000,C 0.000} C_DIS
LIN {X -100.671,Y -271.966,Z 58.905,A 69.687,B 90.000,C 0.000} C_DIS
LIN {X -99.977,Y -270.090,Z 58.905,A 69.687,B 90.000,C 0.000} C_DIS
WAIT SEC 0.1
RET=EKI_SetBool("oxy","torchState",FALSE)
RET = EKI_Send("oxy","torchState")
LIN {X -93.728,Y -253.209,Z 58.905,A 69.687,B 90.000,C 0.000} C_DIS
LIN {X -111.983,Y -245.682,Z 45.730,A 65.496,B 90.000,C 0.000} C_DIS
LIN {X -119.449,Y -262.061,Z 45.730,A 65.496,B 90.000,C 0.000} C_DIS
LIN {X -120.278,Y -263.881,Z 45.730,A 65.496,B 90.000,C 0.000} C_DIS
WAIT SEC 1.75
RET=EKI_SetBool("oxy","torchState",TRUE)
RET = EKI_Send("oxy","torchState")
LIN {X -122.345,Y -262.927,Z 46.762,A 65.046,B 90.000,C 0.000} C_DIS
LIN {X -124.405,Y -261.960,Z 47.797,A 64.597,B 90.000,C 0.000} C_DIS
LIN {X -126.462,Y -260.973,Z 48.818,A 64.146,B 90.000,C 0.000} C_DIS
LIN {X -128.524,Y -259.964,Z 49.808,A 63.693,B 90.000,C 0.000} C_DIS
LIN {X -130.597,Y -258.929,Z 50.746,A 63.235,B 90.000,C 0.000} C_DIS
LIN {X -132.685,Y -257.865,Z 51.615,A 62.772,B 90.000,C 0.000} C_DIS
LIN {X -134.794,Y -256.769,Z 52.391,A 62.302,B 90.000,C 0.000} C_DIS
LIN {X -136.923,Y -255.640,Z 53.055,A 61.826,B 90.000,C 0.000} C_DIS
LIN {X -139.071,Y -254.478,Z 53.585,A 61.344,B 90.000,C 0.000} C_DIS
LIN {X -139.508,Y -254.239,Z 53.676,A 61.245,B 90.000,C 0.000} C_DIS
LIN {X -138.546,Y -252.486,Z 53.676,A 61.245,B 90.000,C 0.000} C_DIS
WAIT SEC 0.1
RET=EKI_SetBool("oxy","torchState",FALSE)
RET = EKI_Send("oxy","torchState")
LIN {X -129.886,Y -236.706,Z 53.676,A 61.245,B 90.000,C 0.000} C_DIS
LIN {X -145.274,Y -227.586,Z 52.101,A 57.449,B 90.000,C 0.000} C_DIS
LIN {X -154.959,Y -242.758,Z 52.101,A 57.449,B 90.000,C 0.000} C_DIS
LIN {X -156.035,Y -244.444,Z 52.101,A 57.449,B 90.000,C 0.000} C_DIS
WAIT SEC 1.75
RET=EKI_SetBool("oxy","torchState",TRUE)
RET = EKI_Send("oxy","torchState")
LIN {X -157.996,Y -243.181,Z 51.202,A 56.988,B 90.000,C 0.000} C_DIS
LIN {X -159.895,Y -241.937,Z 50.155,A 56.540,B 90.000,C 0.000} C_DIS
LIN {X -161.724,Y -240.719,Z 48.964,A 56.105,B 90.000,C 0.000} C_DIS
LIN {X -163.476,Y -239.532,Z 47.634,A 55.687,B 90.000,C 0.000} C_DIS
LIN {X -165.147,Y -238.383,Z 46.171,A 55.287,B 90.000,C 0.000} C_DIS
LIN {X -166.728,Y -237.280,Z 44.580,A 54.906,B 90.000,C 0.000} C_DIS
LIN {X -168.215,Y -236.228,Z 42.868,A 54.546,B 90.000,C 0.000} C_DIS
LIN {X -169.324,Y -235.434,Z 41.430,A 54.276,B 90.000,C 0.000} C_DIS
LIN {X -168.157,Y -233.810,Z 41.430,A 54.276,B 90.000,C 0.000} C_DIS
WAIT SEC 0.1
RET=EKI_SetBool("oxy","torchState",FALSE)
RET = EKI_Send("oxy","torchState")
LIN {X -157.647,Y -219.197,Z 41.430,A 54.276,B 90.000,C 0.000} C_DIS
LIN {X -172.149,Y -208.002,Z 56.028,A 50.388,B 90.000,C 0.000} C_DIS
LIN {X -183.626,Y -221.868,Z 56.028,A 50.388,B 90.000,C 0.000} C_DIS
LIN {X -184.901,Y -223.409,Z 56.028,A 50.388,B 90.000,C 0.000} C_DIS
WAIT SEC 1.75
RET=EKI_SetBool("oxy","torchState",TRUE)
RET = EKI_Send("oxy","torchState")
LIN {X -183.131,Y -224.861,Z 57.032,A 50.840,B 90.000,C 0.000} C_DIS
LIN {X -181.357,Y -226.294,Z 58.055,A 51.291,B 90.000,C 0.000} C_DIS
LIN {X -179.578,Y -227.708,Z 59.096,A 51.740,B 90.000,C 0.000} C_DIS
LIN {X -177.795,Y -229.103,Z 60.156,A 52.187,B 90.000,C 0.000} C_DIS
LIN {X -176.008,Y -230.479,Z 61.235,A 52.632,B 90.000,C 0.000} C_DIS
LIN {X -174.218,Y -231.835,Z 62.331,A 53.076,B 90.000,C 0.000} C_DIS
LIN {X -172.424,Y -233.173,Z 63.446,A 53.518,B 90.000,C 0.000} C_DIS
LIN {X -170.628,Y -234.490,Z 64.580,A 53.958,B 90.000,C 0.000} C_DIS
LIN {X -168.829,Y -235.788,Z 65.734,A 54.397,B 90.000,C 0.000} C_DIS
LIN {X -167.029,Y -237.066,Z 66.905,A 54.833,B 90.000,C 0.000} C_DIS
LIN {X -165.227,Y -238.326,Z 68.094,A 55.267,B 90.000,C 0.000} C_DIS
LIN {X -163.423,Y -239.566,Z 69.301,A 55.700,B 90.000,C 0.000} C_DIS
LIN {X -161.619,Y -240.788,Z 70.526,A 56.130,B 90.000,C 0.000} C_DIS
LIN {X -159.814,Y -241.990,Z 71.769,A 56.559,B 90.000,C 0.000} C_DIS
LIN {X -158.009,Y -243.173,Z 73.030,A 56.985,B 90.000,C 0.000} C_DIS
LIN {X -156.203,Y -244.336,Z 74.310,A 57.409,B 90.000,C 0.000} C_DIS
LIN {X -154.399,Y -245.479,Z 75.608,A 57.831,B 90.000,C 0.000} C_DIS
LIN {X -152.595,Y -246.605,Z 76.923,A 58.251,B 90.000,C 0.000} C_DIS
LIN {X -150.793,Y -247.711,Z 78.256,A 58.669,B 90.000,C 0.000} C_DIS
LIN {X -148.992,Y -248.799,Z 79.606,A 59.085,B 90.000,C 0.000} C_DIS
LIN {X -147.193,Y -249.868,Z 80.973,A 59.498,B 90.000,C 0.000} C_DIS
LIN {X -145.572,Y -250.816,Z 82.222,A 59.869,B 90.000,C 0.000} C_DIS
LIN {X -144.568,Y -249.087,Z 82.222,A 59.869,B 90.000,C 0.000} C_DIS
WAIT SEC 0.1
RET=EKI_SetBool("oxy","torchState",FALSE)
RET = EKI_Send("oxy","torchState")
LIN {X -135.533,Y -233.519,Z 82.222,A 59.869,B 90.000,C 0.000} C_DIS
LIN {X -152.360,Y -222.905,Z 88.884,A 55.647,B 90.000,C 0.000} C_DIS
LIN {X -162.517,Y -237.765,Z 88.884,A 55.647,B 90.000,C 0.000} C_DIS
LIN {X -163.645,Y -239.416,Z 88.884,A 55.647,B 90.000,C 0.000} C_DIS
WAIT SEC 1.75
RET=EKI_SetBool("oxy","torchState",TRUE)
RET = EKI_Send("oxy","torchState")
LIN {X -165.571,Y -238.089,Z 88.001,A 55.185,B 90.000,C 0.000} C_DIS
LIN {X -167.500,Y -236.735,Z 87.169,A 54.719,B 90.000,C 0.000} C_DIS
LIN {X -169.431,Y -235.356,Z 86.381,A 54.250,B 90.000,C 0.000} C_DIS
LIN {X -171.361,Y -233.955,Z 85.632,A 53.779,B 90.000,C 0.000} C_DIS
LIN {X -173.287,Y -232.533,Z 84.915,A 53.306,B 90.000,C 0.000} C_DIS
LIN {X -175.208,Y -231.089,Z 84.226,A 52.831,B 90.000,C 0.000} C_DIS
LIN {X -177.120,Y -229.626,Z 83.555,A 52.355,B 90.000,C 0.000} C_DIS
LIN {X -179.024,Y -228.144,Z 82.898,A 51.879,B 90.000,C 0.000} C_DIS
LIN {X -180.914,Y -226.644,Z 82.248,A 51.402,B 90.000,C 0.000} C_DIS
LIN {X -182.795,Y -225.132,Z 81.596,A 50.925,B 90.000,C 0.000} C_DIS
LIN {X -184.662,Y -223.605,Z 80.939,A 50.449,B 90.000,C 0.000} C_DIS
LIN {X -186.512,Y -222.064,Z 80.269,A 49.973,B 90.000,C 0.000} C_DIS
LIN {X -188.346,Y -220.511,Z 79.580,A 49.498,B 90.000,C 0.000} C_DIS
LIN {X -190.162,Y -218.948,Z 78.866,A 49.025,B 90.000,C 0.000} C_DIS
LIN {X -191.956,Y -217.376,Z 78.118,A 48.554,B 90.000,C 0.000} C_DIS
LIN {X -193.728,Y -215.799,Z 77.332,A 48.085,B 90.000,C 0.000} C_DIS
LIN {X -195.476,Y -214.217,Z 76.501,A 47.619,B 90.000,C 0.000} C_DIS
LIN {X -196.248,Y -213.510,Z 76.115,A 47.412,B 90.000,C 0.000} C_DIS
LIN {X -194.895,Y -212.038,Z 76.115,A 47.412,B 90.000,C 0.000} C_DIS
WAIT SEC 0.1
RET=EKI_SetBool("oxy","torchState",FALSE)
RET = EKI_Send("oxy","torchState")
LIN {X -182.714,Y -198.785,Z 76.115,A 47.412,B 90.000,C 0.000} C_DIS
LIN {X -164.542,Y -214.070,Z 115.744,A 52.453,B 90.000,C 0.000} C_DIS
LIN {X -175.512,Y -228.341,Z 115.744,A 52.453,B 90.000,C 0.000} C_DIS
LIN {X -176.731,Y -229.927,Z 115.744,A 52.453,B 90.000,C 0.000} C_DIS
WAIT SEC 1.75
RET=EKI_SetBool("oxy","torchState",TRUE)
RET = EKI_Send("oxy","torchState")
LIN {X -174.759,Y -231.425,Z 116.082,A 52.942,B 90.000,C 0.000} C_DIS
LIN {X -172.777,Y -232.912,Z 116.416,A 53.432,B 90.000,C 0.000} C_DIS
LIN {X -170.784,Y -234.377,Z 116.776,A 53.920,B 90.000,C 0.000} C_DIS
LIN {X -168.785,Y -235.821,Z 117.187,A 54.407,B 90.000,C 0.000} C_DIS
LIN {X -166.785,Y -237.239,Z 117.675,A 54.892,B 90.000,C 0.000} C_DIS
LIN {X -164.788,Y -238.631,Z 118.240,A 55.373,B 90.000,C 0.000} C_DIS
LIN {X -162.794,Y -239.996,Z 118.881,A 55.850,B 90.000,C 0.000} C_DIS
LIN {X -160.805,Y -241.333,Z 119.592,A 56.324,B 90.000,C 0.000} C_DIS
LIN {X -158.821,Y -242.643,Z 120.364,A 56.793,B 90.000,C 0.000} C_DIS
LIN {X -156.842,Y -243.927,Z 121.192,A 57.259,B 90.000,C 0.000} C_DIS
LIN {X -154.869,Y -245.184,Z 122.071,A 57.722,B 90.000,C 0.000} C_DIS
LIN {X -152.900,Y -246.417,Z 122.994,A 58.181,B 90.000,C 0.000} C_DIS
LIN {X -150.934,Y -247.626,Z 123.954,A 58.637,B 90.000,C 0.000} C_DIS
LIN {X -148.970,Y -248.812,Z 124.948,A 59.090,B 90.000,C 0.000} C_DIS
LIN {X -147.008,Y -249.977,Z 125.966,A 59.541,B 90.000,C 0.000} C_DIS
LIN {X -145.044,Y -251.121,Z 127.007,A 59.990,B 90.000,C 0.000} C_DIS
LIN {X -143.078,Y -252.246,Z 128.064,A 60.437,B 90.000,C 0.000} C_DIS
LIN {X -141.107,Y -253.354,Z 129.131,A 60.884,B 90.000,C 0.000} C_DIS
LIN {X -139.128,Y -254.441,Z 130.204,A 61.330,B 90.000,C 0.000} C_DIS
LIN {X -137.144,Y -255.519,Z 131.276,A 61.776,B 90.000,C 0.000} C_DIS
LIN {X -135.149,Y -256.582,Z 132.344,A 62.223,B 90.000,C 0.000} C_DIS
LIN {X -133.141,Y -257.630,Z 133.402,A 62.670,B 90.000,C 0.000} C_DIS
LIN {X -131.119,Y -258.665,Z 134.444,A 63.119,B 90.000,C 0.000} C_DIS
LIN {X -129.080,Y -259.689,Z 135.466,A 63.570,B 90.000,C 0.000} C_DIS
LIN {X -127.022,Y -260.701,Z 136.460,A 64.023,B 90.000,C 0.000} C_DIS
LIN {X -126.002,Y -261.196,Z 136.942,A 64.247,B 90.000,C 0.000} C_DIS
LIN {X -125.133,Y -259.395,Z 136.942,A 64.247,B 90.000,C 0.000} C_DIS
WAIT SEC 0.1
RET=EKI_SetBool("oxy","torchState",FALSE)
RET = EKI_Send("oxy","torchState")
LIN {X -117.312,Y -243.183,Z 136.942,A 64.247,B 90.000,C 0.000} C_DIS
LIN {X -107.575,Y -247.644,Z 119.972,A 66.520,B 90.000,C 0.000} C_DIS
LIN {X -114.746,Y -264.154,Z 119.972,A 66.520,B 90.000,C 0.000} C_DIS
LIN {X -115.543,Y -265.988,Z 119.972,A 66.520,B 90.000,C 0.000} C_DIS
WAIT SEC 1.75
RET=EKI_SetBool("oxy","torchState",TRUE)
RET = EKI_Send("oxy","torchState")
LIN {X -117.559,Y -265.103,Z 118.789,A 66.085,B 90.000,C 0.000} C_DIS
LIN {X -119.552,Y -264.209,Z 117.573,A 65.654,B 90.000,C 0.000} C_DIS
LIN {X -121.526,Y -263.308,Z 116.333,A 65.225,B 90.000,C 0.000} C_DIS
LIN {X -123.481,Y -262.397,Z 115.069,A 64.799,B 90.000,C 0.000} C_DIS
LIN {X -125.418,Y -261.477,Z 113.785,A 64.375,B 90.000,C 0.000} C_DIS
LIN {X -127.339,Y -260.547,Z 112.484,A 63.953,B 90.000,C 0.000} C_DIS
LIN {X -129.247,Y -259.606,Z 111.170,A 63.533,B 90.000,C 0.000} C_DIS
LIN {X -131.141,Y -258.653,Z 109.846,A 63.114,B 90.000,C 0.000} C_DIS
LIN {X -133.024,Y -257.688,Z 108.516,A 62.696,B 90.000,C 0.000} C_DIS
LIN {X -134.901,Y -256.711,Z 107.184,A 62.278,B 90.000,C 0.000} C_DIS
LIN {X -136.769,Y -255.719,Z 105.852,A 61.860,B 90.000,C 0.000} C_DIS
LIN {X -138.633,Y -254.714,Z 104.524,A 61.442,B 90.000,C 0.000} C_DIS
LIN {X -139.860,Y -254.046,Z 103.651,A 61.166,B 90.000,C 0.000} C_DIS
LIN {X -138.895,Y -252.294,Z 103.651,A 61.166,B 90.000,C 0.000} C_DIS
WAIT SEC 0.1
RET=EKI_SetBool("oxy","torchState",FALSE)
RET = EKI_Send("oxy","torchState")
LIN {X -130.214,Y -236.525,Z 103.651,A 61.166,B 90.000,C 0.000} C_DIS
LIN {X -117.104,Y -243.283,Z 92.160,A 64.296,B 90.000,C 0.000} C_DIS
LIN {X -124.911,Y -259.502,Z 92.160,A 64.296,B 90.000,C 0.000} C_DIS
LIN {X -125.779,Y -261.304,Z 92.160,A 64.296,B 90.000,C 0.000} C_DIS
WAIT SEC 1.75
RET=EKI_SetBool("oxy","torchState",TRUE)
RET = EKI_Send("oxy","torchState")
LIN {X -123.523,Y -262.377,Z 92.069,A 64.790,B 90.000,C 0.000} C_DIS
LIN {X -121.290,Y -263.418,Z 91.647,A 65.276,B 90.000,C 0.000} C_DIS
LIN {X -119.128,Y -264.402,Z 90.869,A 65.746,B 90.000,C 0.000} C_DIS
LIN {X -117.100,Y -265.306,Z 89.719,A 66.184,B 90.000,C 0.000} C_DIS
LIN {X -115.250,Y -266.115,Z 88.246,A 66.583,B 90.000,C 0.000} C_DIS
LIN {X -113.592,Y -266.827,Z 86.516,A 66.940,B 90.000,C 0.000} C_DIS
LIN {X -112.127,Y -267.446,Z 84.588,A 67.254,B 90.000,C 0.000} C_DIS
LIN {X -112.003,Y -267.498,Z 84.405,A 67.281,B 90.000,C 0.000} C_DIS
LIN {X -111.230,Y -265.654,Z 84.405,A 67.281,B 90.000,C 0.000} C_DIS
WAIT SEC 0.1
RET=EKI_SetBool("oxy","torchState",FALSE)
RET = EKI_Send("oxy","torchState")
LIN {X -104.278,Y -249.050,Z 84.405,A 67.281,B 90.000,C 0.000} C_DIS
LIN {X -52.771,Y -264.793,Z 52.150,A 78.729,B 90.000,C 0.000} C_DIS
LIN {X -56.289,Y -282.446,Z 52.150,A 78.729,B 90.000,C 0.000} C_DIS
LIN {X -56.680,Y -284.407,Z 52.150,A 78.729,B 90.000,C 0.000} C_DIS
WAIT SEC 1.75
RET=EKI_SetBool("oxy","torchState",TRUE)
RET = EKI_Send("oxy","torchState")
LIN {X -54.305,Y -284.870,Z 51.525,A 79.207,B 90.000,C 0.000} C_DIS
LIN {X -51.893,Y -285.319,Z 51.044,A 79.692,B 90.000,C 0.000} C_DIS
LIN {X -49.458,Y -285.751,Z 50.681,A 80.181,B 90.000,C 0.000} C_DIS
LIN {X -47.008,Y -286.165,Z 50.408,A 80.671,B 90.000,C 0.000} C_DIS
LIN {X -44.548,Y -286.558,Z 50.196,A 81.164,B 90.000,C 0.000} C_DIS
LIN {X -42.083,Y -286.929,Z 50.015,A 81.656,B 90.000,C 0.000} C_DIS
LIN {X -39.614,Y -287.281,Z 49.836,A 82.149,B 90.000,C 0.000} C_DIS
LIN {X -37.145,Y -287.611,Z 49.634,A 82.641,B 90.000,C 0.000} C_DIS
LIN {X -34.678,Y -287.919,Z 49.375,A 83.132,B 90.000,C 0.000} C_DIS
LIN {X -32.218,Y -288.205,Z 49.037,A 83.622,B 90.000,C 0.000} C_DIS
LIN {X -29.772,Y -288.467,Z 48.591,A 84.107,B 90.000,C 0.000} C_DIS
LIN {X -27.344,Y -288.708,Z 48.049,A 84.590,B 90.000,C 0.000} C_DIS
LIN {X -24.932,Y -288.926,Z 47.428,A 85.068,B 90.000,C 0.000} C_DIS
LIN {X -22.537,Y -289.123,Z 46.742,A 85.543,B 90.000,C 0.000} C_DIS
LIN {X -20.153,Y -289.298,Z 46.009,A 86.015,B 90.000,C 0.000} C_DIS
LIN {X -17.777,Y -289.454,Z 45.248,A 86.486,B 90.000,C 0.000} C_DIS
LIN {X -15.405,Y -289.590,Z 44.473,A 86.955,B 90.000,C 0.000} C_DIS
LIN {X -13.031,Y -289.706,Z 43.699,A 87.425,B 90.000,C 0.000} C_DIS
LIN {X -12.459,Y -289.732,Z 43.514,A 87.538,B 90.000,C 0.000} C_DIS
LIN {X -12.374,Y -287.734,Z 43.514,A 87.538,B 90.000,C 0.000} C_DIS
WAIT SEC 0.1
RET=EKI_SetBool("oxy","torchState",FALSE)
RET = EKI_Send("oxy","torchState")
LIN {X -11.600,Y -269.751,Z 43.514,A 87.538,B 90.000,C 0.000} C_DIS
LIN {X -10.649,Y -269.790,Z 60.571,A 87.740,B 90.000,C 0.000} C_DIS
LIN {X -11.359,Y -287.776,Z 60.571,A 87.740,B 90.000,C 0.000} C_DIS
LIN {X -11.437,Y -289.774,Z 60.571,A 87.740,B 90.000,C 0.000} C_DIS
WAIT SEC 1.75
RET=EKI_SetBool("oxy","torchState",TRUE)
RET = EKI_Send("oxy","torchState")
LIN {X -13.928,Y -289.665,Z 60.756,A 87.247,B 90.000,C 0.000} C_DIS
LIN {X -16.408,Y -289.535,Z 61.037,A 86.756,B 90.000,C 0.000} C_DIS
LIN {X -18.876,Y -289.385,Z 61.409,A 86.268,B 90.000,C 0.000} C_DIS
LIN {X -21.325,Y -289.214,Z 61.877,A 85.783,B 90.000,C 0.000} C_DIS
LIN {X -23.754,Y -289.025,Z 62.439,A 85.302,B 90.000,C 0.000} C_DIS
LIN {X -26.156,Y -288.818,Z 63.097,A 84.825,B 90.000,C 0.000} C_DIS
LIN {X -28.529,Y -288.593,Z 63.850,A 84.354,B 90.000,C 0.000} C_DIS
LIN {X -30.867,Y -288.352,Z 64.702,A 83.890,B 90.000,C 0.000} C_DIS
LIN {X -33.166,Y -288.097,Z 65.649,A 83.433,B 90.000,C 0.000} C_DIS
LIN {X -35.419,Y -287.829,Z 66.698,A 82.985,B 90.000,C 0.000} C_DIS
LIN {X -37.623,Y -287.549,Z 67.843,A 82.546,B 90.000,C 0.000} C_DIS
LIN {X -39.772,Y -287.260,Z 69.088,A 82.117,B 90.000,C 0.000} C_DIS
LIN {X -41.858,Y -286.963,Z 70.432,A 81.701,B 90.000,C 0.000} C_DIS
LIN {X -43.878,Y -286.661,Z 71.873,A 81.298,B 90.000,C 0.000} C_DIS
LIN {X -45.057,Y -286.478,Z 72.784,A 81.062,B 90.000,C 0.000} C_DIS
LIN {X -44.746,Y -284.503,Z 72.784,A 81.062,B 90.000,C 0.000} C_DIS
WAIT SEC 0.1
RET=EKI_SetBool("oxy","torchState",FALSE)
RET = EKI_Send("oxy","torchState")
LIN {X -41.950,Y -266.721,Z 72.784,A 81.062,B 90.000,C 0.000} C_DIS
LIN {X -6.678,Y -269.917,Z 78.844,A 88.583,B 90.000,C 0.000} C_DIS
LIN {X -7.123,Y -287.912,Z 78.844,A 88.583,B 90.000,C 0.000} C_DIS
LIN {X -7.173,Y -289.911,Z 78.844,A 88.583,B 90.000,C 0.000} C_DIS
WAIT SEC 1.75
RET=EKI_SetBool("oxy","torchState",TRUE)
RET = EKI_Send("oxy","torchState")
LIN {X -5.314,Y -289.951,Z 77.173,A 88.950,B 90.000,C 0.000} C_DIS
LIN {X -3.186,Y -289.982,Z 75.861,A 89.370,B 90.000,C 0.000} C_DIS
LIN {X -0.875,Y -289.999,Z 74.910,A 89.827,B 90.000,C 0.000} C_DIS
LIN {X 1.552,Y -289.996,Z 74.309,A 90.307,B 90.000,C 0.000} C_DIS
LIN {X 4.037,Y -289.972,Z 74.039,A 90.798,B 90.000,C 0.000} C_DIS
LIN {X 6.536,Y -289.926,Z 74.059,A 91.291,B 90.000,C 0.000} C_DIS
LIN {X 9.020,Y -289.860,Z 74.329,A 91.782,B 90.000,C 0.000} C_DIS
LIN {X 11.207,Y -289.783,Z 74.744,A 92.215,B 90.000,C 0.000} C_DIS
LIN {X 11.130,Y -287.785,Z 74.744,A 92.215,B 90.000,C 0.000} C_DIS
WAIT SEC 0.1
RET=EKI_SetBool("oxy","torchState",FALSE)
RET = EKI_Send("oxy","torchState")
LIN {X 10.435,Y -269.798,Z 74.744,A 92.215,B 90.000,C 0.000} C_DIS
LIN {X 3.278,Y -269.980,Z 60.571,A 90.696,B 90.000,C 0.000} C_DIS
LIN {X 3.497,Y -287.979,Z 60.571,A 90.696,B 90.000,C 0.000} C_DIS
LIN {X 3.521,Y -289.979,Z 60.571,A 90.696,B 90.000,C 0.000} C_DIS
WAIT SEC 1.75
RET=EKI_SetBool("oxy","torchState",TRUE)
RET = EKI_Send("oxy","torchState")
LIN {X 6.020,Y -289.936,Z 60.559,A 91.189,B 90.000,C 0.000} C_DIS
LIN {X 8.519,Y -289.875,Z 60.514,A 91.683,B 90.000,C 0.000} C_DIS
LIN {X 11.015,Y -289.789,Z 60.432,A 92.177,B 90.000,C 0.000} C_DIS
LIN {X 13.511,Y -289.685,Z 60.322,A 92.670,B 90.000,C 0.000} C_DIS
LIN {X 16.003,Y -289.557,Z 60.180,A 93.163,B 90.000,C 0.000} C_DIS
LIN {X 18.493,Y -289.408,Z 60.013,A 93.656,B 90.000,C 0.000} C_DIS
LIN {X 20.979,Y -289.238,Z 59.825,A 94.149,B 90.000,C 0.000} C_DIS
LIN {X 23.463,Y -289.048,Z 59.616,A 94.641,B 90.000,C 0.000} C_DIS
LIN {X 25.944,Y -288.836,Z 59.390,A 95.133,B 90.000,C 0.000} C_DIS
LIN {X 28.421,Y -288.602,Z 59.149,A 95.624,B 90.000,C 0.000} C_DIS
LIN {X 30.894,Y -288.346,Z 58.897,A 96.116,B 90.000,C 0.000} C_DIS
LIN {X 33.365,Y -288.069,Z 58.636,A 96.607,B 90.000,C 0.000} C_DIS
LIN {X 35.833,Y -287.776,Z 58.370,A 97.098,B 90.000,C 0.000} C_DIS
LIN {X 38.298,Y -287.460,Z 58.101,A 97.589,B 90.000,C 0.000} C_DIS
LIN {X 40.760,Y -287.121,Z 57.831,A 98.080,B 90.000,C 0.000} C_DIS
LIN {X 43.219,Y -286.757,Z 57.564,A 98.571,B 90.000,C 0.000} C_DIS
LIN {X 45.675,Y -286.379,Z 57.301,A 99.062,B 90.000,C 0.000} C_DIS
LIN {X 48.130,Y -285.978,Z 57.047,A 99.553,B 90.000,C 0.000} C_DIS
LIN {X 50.581,Y -285.554,Z 56.803,A 100.045,B 90.000,C 0.000} C_DIS
LIN {X 53.030,Y -285.109,Z 56.574,A 100.537,B 90.000,C 0.000} C_DIS
LIN {X 53.535,Y -285.016,Z 56.527,A 100.638,B 90.000,C 0.000} C_DIS
LIN {X 53.166,Y -283.050,Z 56.527,A 100.638,B 90.000,C 0.000} C_DIS
WAIT SEC 0.1
RET=EKI_SetBool("oxy","torchState",FALSE)
RET = EKI_Send("oxy","torchState")
LIN {X 49.843,Y -265.359,Z 56.527,A 100.638,B 90.000,C 0.000} C_DIS
LIN {X 67.865,Y -261.332,Z 83.554,A 104.557,B 90.000,C 0.000} C_DIS
LIN {X 72.389,Y -278.754,Z 83.554,A 104.557,B 90.000,C 0.000} C_DIS
LIN {X 72.892,Y -280.690,Z 83.554,A 104.557,B 90.000,C 0.000} C_DIS
WAIT SEC 1.75
RET=EKI_SetBool("oxy","torchState",TRUE)
RET = EKI_Send("oxy","torchState")
LIN {X 70.477,Y -281.305,Z 83.361,A 104.065,B 90.000,C 0.000} C_DIS
LIN {X 68.052,Y -281.901,Z 83.239,A 103.572,B 90.000,C 0.000} C_DIS
LIN {X 65.621,Y -282.477,Z 83.178,A 103.078,B 90.000,C 0.000} C_DIS
LIN {X 63.184,Y -283.033,Z 83.164,A 102.584,B 90.000,C 0.000} C_DIS
LIN {X 60.742,Y -283.567,Z 83.186,A 102.090,B 90.000,C 0.000} C_DIS
LIN {X 58.296,Y -284.080,Z 83.230,A 101.597,B 90.000,C 0.000} C_DIS
LIN {X 55.845,Y -284.571,Z 83.285,A 101.103,B 90.000,C 0.000} C_DIS
LIN {X 53.391,Y -285.043,Z 83.338,A 100.609,B 90.000,C 0.000} C_DIS
LIN {X 50.932,Y -285.491,Z 83.374,A 100.115,B 90.000,C 0.000} C_DIS
LIN {X 48.469,Y -285.920,Z 83.385,A 99.621,B 90.000,C 0.000} C_DIS
LIN {X 46.003,Y -286.327,Z 83.355,A 99.128,B 90.000,C 0.000} C_DIS
LIN {X 43.535,Y -286.713,Z 83.272,A 98.634,B 90.000,C 0.000} C_DIS
LIN {X 41.066,Y -287.077,Z 83.123,A 98.141,B 90.000,C 0.000} C_DIS
LIN {X 38.601,Y -287.419,Z 82.894,A 97.649,B 90.000,C 0.000} C_DIS
LIN {X 36.143,Y -287.739,Z 82.570,A 97.159,B 90.000,C 0.000} C_DIS
LIN {X 33.698,Y -288.035,Z 82.141,A 96.673,B 90.000,C 0.000} C_DIS
LIN {X 31.274,Y -288.309,Z 81.595,A 96.191,B 90.000,C 0.000} C_DIS
LIN {X 29.801,Y -288.465,Z 81.199,A 95.898,B 90.000,C 0.000} C_DIS
LIN {X 29.596,Y -286.475,Z 81.199,A 95.898,B 90.000,C 0.000} C_DIS
WAIT SEC 0.1
RET=EKI_SetBool("oxy","torchState",FALSE)
RET = EKI_Send("oxy","torchState")
LIN {X 27.746,Y -268.571,Z 81.199,A 95.898,B 90.000,C 0.000} C_DIS
LIN {X 26.805,Y -268.666,Z 101.898,A 95.698,B 90.000,C 0.000} C_DIS
LIN {X 28.592,Y -286.577,Z 101.898,A 95.698,B 90.000,C 0.000} C_DIS
LIN {X 28.791,Y -288.567,Z 101.898,A 95.698,B 90.000,C 0.000} C_DIS
WAIT SEC 1.75
RET=EKI_SetBool("oxy","torchState",TRUE)
RET = EKI_Send("oxy","torchState")
LIN {X 31.267,Y -288.309,Z 102.124,A 96.189,B 90.000,C 0.000} C_DIS
LIN {X 33.723,Y -288.033,Z 102.499,A 96.678,B 90.000,C 0.000} C_DIS
LIN {X 36.150,Y -287.738,Z 103.016,A 97.161,B 90.000,C 0.000} C_DIS
LIN {X 38.543,Y -287.427,Z 103.670,A 97.638,B 90.000,C 0.000} C_DIS
LIN {X 40.894,Y -287.102,Z 104.455,A 98.106,B 90.000,C 0.000} C_DIS
LIN {X 43.198,Y -286.764,Z 105.364,A 98.567,B 90.000,C 0.000} C_DIS
LIN {X 45.452,Y -286.416,Z 106.388,A 99.017,B 90.000,C 0.000} C_DIS
LIN {X 47.651,Y -286.058,Z 107.521,A 99.457,B 90.000,C 0.000} C_DIS
LIN {X 49.792,Y -285.693,Z 108.759,A 99.886,B 90.000,C 0.000} C_DIS
LIN {X 51.870,Y -285.323,Z 110.097,A 100.304,B 90.000,C 0.000} C_DIS
LIN {X 53.886,Y -284.949,Z 111.527,A 100.709,B 90.000,C 0.000} C_DIS
LIN {X 55.835,Y -284.574,Z 113.046,A 101.101,B 90.000,C 0.000} C_DIS
LIN {X 56.693,Y -284.405,Z 113.760,A 101.273,B 90.000,C 0.000} C_DIS
LIN {X 56.302,Y -282.443,Z 113.760,A 101.273,B 90.000,C 0.000} C_DIS
WAIT SEC 0.1
RET=EKI_SetBool("oxy","torchState",FALSE)
RET = EKI_Send("oxy","torchState")
LIN {X 52.783,Y -264.790,Z 113.760,A 101.273,B 90.000,C 0.000} C_DIS
LIN {X 69.970,Y -260.776,Z 138.204,A 105.020,B 90.000,C 0.000} C_DIS
LIN {X 74.635,Y -278.161,Z 138.204,A 105.020,B 90.000,C 0.000} C_DIS
LIN {X 75.153,Y -280.093,Z 138.204,A 105.020,B 90.000,C 0.000} C_DIS
WAIT SEC 1.75
RET=EKI_SetBool("oxy","torchState",TRUE)
RET = EKI_Send("oxy","torchState")
LIN {X 76.251,Y -279.796,Z 140.431,A 105.244,B 90.000,C 0.000} C_DIS
LIN {X 77.296,Y -279.509,Z 142.683,A 105.458,B 90.000,C 0.000} C_DIS
LIN {X 78.283,Y -279.234,Z 144.963,A 105.661,B 90.000,C 0.000} C_DIS
LIN {X 79.208,Y -278.973,Z 147.271,A 105.851,B 90.000,C 0.000} C_DIS
LIN {X 80.065,Y -278.728,Z 149.606,A 106.027,B 90.000,C 0.000} C_DIS
LIN {X 80.851,Y -278.502,Z 151.968,A 106.188,B 90.000,C 0.000} C_DIS
LIN {X 81.555,Y -278.296,Z 154.358,A 106.333,B 90.000,C 0.000} C_DIS
LIN {X 82.177,Y -278.113,Z 156.772,A 106.461,B 90.000,C 0.000} C_DIS
LIN {X 82.708,Y -277.956,Z 159.210,A 106.571,B 90.000,C 0.000} C_DIS
LIN {X 83.142,Y -277.826,Z 161.668,A 106.660,B 90.000,C 0.000} C_DIS
LIN {X 83.472,Y -277.727,Z 164.144,A 106.728,B 90.000,C 0.000} C_DIS
LIN {X 83.695,Y -277.660,Z 166.632,A 106.774,B 90.000,C 0.000} C_DIS
LIN {X 83.804,Y -277.627,Z 169.130,A 106.797,B 90.000,C 0.000} C_DIS
LIN {X 83.226,Y -275.712,Z 169.130,A 106.797,B 90.000,C 0.000} C_DIS
WAIT SEC 0.1
RET=EKI_SetBool("oxy","torchState",FALSE)
RET = EKI_Send("oxy","torchState")
LIN {X 78.025,Y -258.480,Z 169.130,A 106.797,B 90.000,C 0.000} C_DIS
LIN {X 95.918,Y -252.388,Z 187.497,A 110.809,B 90.000,C 0.000} C_DIS
LIN {X 102.313,Y -269.214,Z 187.497,A 110.809,B 90.000,C 0.000} C_DIS
LIN {X 103.023,Y -271.083,Z 187.497,A 110.809,B 90.000,C 0.000} C_DIS
WAIT SEC 1.75
RET=EKI_SetBool("oxy","torchState",TRUE)
RET = EKI_Send("oxy","torchState")
LIN {X 102.516,Y -271.276,Z 189.938,A 110.702,B 90.000,C 0.000} C_DIS
LIN {X 101.946,Y -271.491,Z 192.362,A 110.581,B 90.000,C 0.000} C_DIS
LIN {X 101.307,Y -271.729,Z 194.767,A 110.447,B 90.000,C 0.000} C_DIS
LIN {X 100.601,Y -271.991,Z 197.151,A 110.298,B 90.000,C 0.000} C_DIS
LIN {X 99.826,Y -272.277,Z 199.510,A 110.135,B 90.000,C 0.000} C_DIS
LIN {X 98.981,Y -272.585,Z 201.842,A 109.957,B 90.000,C 0.000} C_DIS
LIN {X 98.062,Y -272.917,Z 204.143,A 109.764,B 90.000,C 0.000} C_DIS
LIN {X 97.067,Y -273.273,Z 206.409,A 109.555,B 90.000,C 0.000} C_DIS
LIN {X 95.998,Y -273.650,Z 208.636,A 109.331,B 90.000,C 0.000} C_DIS
LIN {X 94.849,Y -274.050,Z 210.820,A 109.091,B 90.000,C 0.000} C_DIS
LIN {X 93.621,Y -274.472,Z 212.956,A 108.834,B 90.000,C 0.000} C_DIS
LIN {X 92.313,Y -274.915,Z 215.039,A 108.561,B 90.000,C 0.000} C_DIS
LIN {X 90.923,Y -275.378,Z 217.065,A 108.272,B 90.000,C 0.000} C_DIS
LIN {X 89.450,Y -275.860,Z 219.026,A 107.966,B 90.000,C 0.000} C_DIS
LIN {X 88.505,Y -276.165,Z 220.202,A 107.770,B 90.000,C 0.000} C_DIS
LIN {X 87.894,Y -274.260,Z 220.202,A 107.770,B 90.000,C 0.000} C_DIS
WAIT SEC 0.1
RET=EKI_SetBool("oxy","torchState",FALSE)
RET = EKI_Send("oxy","torchState")
LIN {X 82.401,Y -257.119,Z 220.202,A 107.770,B 90.000,C 0.000} C_DIS
LIN {X 63.077,Y -262.529,Z 209.016,A 103.510,B 90.000,C 0.000} C_DIS
LIN {X 67.282,Y -280.031,Z 209.016,A 103.510,B 90.000,C 0.000} C_DIS
LIN {X 67.749,Y -281.975,Z 209.016,A 103.510,B 90.000,C 0.000} C_DIS
WAIT SEC 1.75
RET=EKI_SetBool("oxy","torchState",TRUE)
RET = EKI_Send("oxy","torchState")
LIN {X 65.995,Y -282.391,Z 210.748,A 103.154,B 90.000,C 0.000} C_DIS
LIN {X 64.171,Y -282.811,Z 212.405,A 102.784,B 90.000,C 0.000} C_DIS
LIN {X 62.281,Y -283.233,Z 213.986,A 102.402,B 90.000,C 0.000} C_DIS
LIN {X 60.329,Y -283.655,Z 215.488,A 102.007,B 90.000,C 0.000} C_DIS
LIN {X 58.318,Y -284.076,Z 216.912,A 101.601,B 90.000,C 0.000} C_DIS
LIN {X 56.252,Y -284.492,Z 218.256,A 101.185,B 90.000,C 0.000} C_DIS
LIN {X 54.136,Y -284.902,Z 219.522,A 100.759,B 90.000,C 0.000} C_DIS
LIN {X 51.970,Y -285.305,Z 220.704,A 100.324,B 90.000,C 0.000} C_DIS
LIN {X 49.763,Y -285.698,Z 221.809,A 99.881,B 90.000,C 0.000} C_DIS
LIN {X 47.514,Y -286.081,Z 222.832,A 99.430,B 90.000,C 0.000} C_DIS
LIN {X 45.228,Y -286.451,Z 223.773,A 98.972,B 90.000,C 0.000} C_DIS
LIN {X 42.909,Y -286.808,Z 224.635,A 98.509,B 90.000,C 0.000} C_DIS
LIN {X 40.559,Y -287.150,Z 225.416,A 98.040,B 90.000,C 0.000} C_DIS
LIN {X 38.181,Y -287.475,Z 226.114,A 97.566,B 90.000,C 0.000} C_DIS
LIN {X 35.779,Y -287.784,Z 226.732,A 97.087,B 90.000,C 0.000} C_DIS
LIN {X 33.355,Y -288.075,Z 227.270,A 96.605,B 90.000,C 0.000} C_DIS
LIN {X 30.912,Y -288.347,Z 227.723,A 96.119,B 90.000,C 0.000} C_DIS
LIN {X 29.049,Y -288.541,Z 228.014,A 95.749,B 90.000,C 0.000} C_DIS
LIN {X 28.849,Y -286.551,Z 228.014,A 95.749,B 90.000,C 0.000} C_DIS
WAIT SEC 0.1
RET=EKI_SetBool("oxy","torchState",FALSE)
RET = EKI_Send("oxy","torchState")
LIN {X 27.046,Y -268.642,Z 228.014,A 95.749,B 90.000,C 0.000} C_DIS
LIN {X -5.272,Y -269.949,Z 225.659,A 88.881,B 90.000,C 0.000} C_DIS
LIN {X -5.623,Y -287.945,Z 225.659,A 88.881,B 90.000,C 0.000} C_DIS
LIN {X -5.662,Y -289.945,Z 225.659,A 88.881,B 90.000,C 0.000} C_DIS
WAIT SEC 1.75
RET=EKI_SetBool("oxy","torchState",TRUE)
RET = EKI_Send("oxy","torchState")
LIN {X -8.069,Y -289.888,Z 224.985,A 88.406,B 90.000,C 0.000} C_DIS
LIN {X -10.461,Y -289.811,Z 224.264,A 87.933,B 90.000,C 0.000} C_DIS
LIN {X -12.841,Y -289.715,Z 223.507,A 87.462,B 90.000,C 0.000} C_DIS
LIN {X -15.213,Y -289.600,Z 222.726,A 86.993,B 90.000,C 0.000} C_DIS
LIN {X -17.580,Y -289.464,Z 221.933,A 86.525,B 90.000,C 0.000} C_DIS
LIN {X -19.946,Y -289.311,Z 221.142,A 86.056,B 90.000,C 0.000} C_DIS
LIN {X -22.314,Y -289.140,Z 220.361,A 85.587,B 90.000,C 0.000} C_DIS
LIN {X -24.689,Y -288.946,Z 219.605,A 85.116,B 90.000,C 0.000} C_DIS
LIN {X -27.073,Y -288.733,Z 218.884,A 84.643,B 90.000,C 0.000} C_DIS
LIN {X -29.469,Y -288.499,Z 218.212,A 84.168,B 90.000,C 0.000} C_DIS
LIN {X -31.880,Y -288.242,Z 217.603,A 83.689,B 90.000,C 0.000} C_DIS
LIN {X -34.306,Y -287.963,Z 217.070,A 83.206,B 90.000,C 0.000} C_DIS
LIN {X -36.747,Y -287.662,Z 216.622,A 82.720,B 90.000,C 0.000} C_DIS
LIN {X -39.202,Y -287.338,Z 216.278,A 82.231,B 90.000,C 0.000} C_DIS
LIN {X -41.666,Y -286.991,Z 216.040,A 81.739,B 90.000,C 0.000} C_DIS
LIN {X -44.133,Y -286.622,Z 215.878,A 81.247,B 90.000,C 0.000} C_DIS
LIN {X -46.598,Y -286.231,Z 215.743,A 80.753,B 90.000,C 0.000} C_DIS
LIN {X -49.059,Y -285.820,Z 215.590,A 80.261,B 90.000,C 0.000} C_DIS
LIN {X -50.740,Y -285.527,Z 215.452,A 79.923,B 90.000,C 0.000} C_DIS
LIN {X -50.390,Y -283.558,Z 215.452,A 79.923,B 90.000,C 0.000} C_DIS
WAIT SEC 0.1
RET=EKI_SetBool("oxy","torchState",FALSE)
RET = EKI_Send("oxy","torchState")
LIN {X -47.240,Y -265.835,Z 215.452,A 79.923,B 90.000,C 0.000} C_DIS
LIN {X -137.250,Y -232.513,Z 153.837,A 59.447,B 90.000,C 0.000} C_DIS
LIN {X -146.400,Y -248.014,Z 153.837,A 59.447,B 90.000,C 0.000} C_DIS
LIN {X -147.417,Y -249.737,Z 153.837,A 59.447,B 90.000,C 0.000} C_DIS
WAIT SEC 1.75
RET=EKI_SetBool("oxy","torchState",TRUE)
RET = EKI_Send("oxy","torchState")
LIN {X -149.357,Y -248.579,Z 152.766,A 59.001,B 90.000,C 0.000} C_DIS
LIN {X -151.288,Y -247.404,Z 151.700,A 58.554,B 90.000,C 0.000} C_DIS
LIN {X -153.215,Y -246.219,Z 150.637,A 58.107,B 90.000,C 0.000} C_DIS
LIN {X -155.135,Y -245.016,Z 149.581,A 57.660,B 90.000,C 0.000} C_DIS
LIN {X -157.048,Y -243.793,Z 148.534,A 57.211,B 90.000,C 0.000} C_DIS
LIN {X -158.955,Y -242.554,Z 147.498,A 56.762,B 90.000,C 0.000} C_DIS
LIN {X -160.857,Y -241.296,Z 146.474,A 56.311,B 90.000,C 0.000} C_DIS
LIN {X -162.755,Y -240.021,Z 145.464,A 55.859,B 90.000,C 0.000} C_DIS
LIN {X -164.648,Y -238.727,Z 144.469,A 55.406,B 90.000,C 0.000} C_DIS
LIN {X -166.538,Y -237.413,Z 143.492,A 54.952,B 90.000,C 0.000} C_DIS
LIN {X -168.029,Y -236.361,Z 142.734,A 54.591,B 90.000,C 0.000} C_DIS
LIN {X -166.870,Y -234.731,Z 142.734,A 54.591,B 90.000,C 0.000} C_DIS
WAIT SEC 0.1
RET=EKI_SetBool("oxy","torchState",FALSE)
RET = EKI_Send("oxy","torchState")
LIN {X -156.441,Y -220.060,Z 142.734,A 54.591,B 90.000,C 0.000} C_DIS
LIN {X -215.842,Y -162.211,Z 92.190,A 36.926,B 90.000,C 0.000} C_DIS
LIN {X -230.231,Y -173.025,Z 92.190,A 36.926,B 90.000,C 0.000} C_DIS
LIN {X -231.830,Y -174.226,Z 92.190,A 36.926,B 90.000,C 0.000} C_DIS
WAIT SEC 1.75
RET=EKI_SetBool("oxy","torchState",TRUE)
RET = EKI_Send("oxy","torchState")
LIN {X -233.204,Y -172.379,Z 91.218,A 36.471,B 90.000,C 0.000} C_DIS
LIN {X -234.565,Y -170.521,Z 90.245,A 36.016,B 90.000,C 0.000} C_DIS
LIN {X -235.913,Y -168.652,Z 89.276,A 35.561,B 90.000,C 0.000} C_DIS
LIN {X -237.249,Y -166.769,Z 88.320,A 35.104,B 90.000,C 0.000} C_DIS
LIN {X -238.575,Y -164.869,Z 87.381,A 34.647,B 90.000,C 0.000} C_DIS
LIN {X -239.890,Y -162.948,Z 86.470,A 34.187,B 90.000,C 0.000} C_DIS
LIN {X -241.198,Y -161.008,Z 85.590,A 33.724,B 90.000,C 0.000} C_DIS
LIN {X -242.497,Y -159.043,Z 84.753,A 33.259,B 90.000,C 0.000} C_DIS
LIN {X -243.790,Y -157.055,Z 83.964,A 32.791,B 90.000,C 0.000} C_DIS
LIN {X -245.076,Y -155.041,Z 83.230,A 32.318,B 90.000,C 0.000} C_DIS
LIN {X -245.937,Y -153.672,Z 82.769,A 31.999,B 90.000,C 0.000} C_DIS
LIN {X -244.241,Y -152.612,Z 82.769,A 31.999,B 90.000,C 0.000} C_DIS
WAIT SEC 0.1
RET=EKI_SetBool("oxy","torchState",FALSE)
RET = EKI_Send("oxy","torchState")
LIN {X -228.976,Y -143.074,Z 82.769,A 31.999,B 90.000,C 0.000} C_DIS
LIN {X -231.316,Y -139.258,Z 52.244,A 31.049,B 90.000,C 0.000} C_DIS
LIN {X -246.737,Y -148.542,Z 52.244,A 31.049,B 90.000,C 0.000} C_DIS
LIN {X -248.451,Y -149.574,Z 52.244,A 31.049,B 90.000,C 0.000} C_DIS
WAIT SEC 1.75
RET=EKI_SetBool("oxy","torchState",TRUE)
RET = EKI_Send("oxy","torchState")
LIN {X -247.180,Y -151.664,Z 52.757,A 31.532,B 90.000,C 0.000} C_DIS
LIN {X -245.900,Y -153.730,Z 53.345,A 32.012,B 90.000,C 0.000} C_DIS
LIN {X -244.609,Y -155.776,Z 53.973,A 32.490,B 90.000,C 0.000} C_DIS
LIN {X -243.302,Y -157.810,Z 54.608,A 32.968,B 90.000,C 0.000} C_DIS
LIN {X -241.974,Y -159.839,Z 55.216,A 33.447,B 90.000,C 0.000} C_DIS
LIN {X -240.621,Y -161.869,Z 55.760,A 33.929,B 90.000,C 0.000} C_DIS
LIN {X -239.239,Y -163.904,Z 56.204,A 34.415,B 90.000,C 0.000} C_DIS
LIN {X -237.830,Y -165.942,Z 56.533,A 34.905,B 90.000,C 0.000} C_DIS
LIN {X -236.397,Y -167.976,Z 56.770,A 35.396,B 90.000,C 0.000} C_DIS
LIN {X -234.944,Y -170.002,Z 56.952,A 35.889,B 90.000,C 0.000} C_DIS
LIN {X -233.473,Y -172.017,Z 57.109,A 36.382,B 90.000,C 0.000} C_DIS
LIN {X -231.985,Y -174.019,Z 57.274,A 36.875,B 90.000,C 0.000} C_DIS
LIN {X -230.482,Y -176.006,Z 57.479,A 37.367,B 90.000,C 0.000} C_DIS
LIN {X -228.966,Y -177.973,Z 57.760,A 37.858,B 90.000,C 0.000} C_DIS
LIN {X -228.800,Y -178.187,Z 57.795,A 37.911,B 90.000,C 0.000} C_DIS
LIN {X -227.222,Y -176.958,Z 57.795,A 37.911,B 90.000,C 0.000} C_DIS
WAIT SEC 0.1
RET=EKI_SetBool("oxy","torchState",FALSE)
RET = EKI_Send("oxy","torchState")
LIN {X -213.021,Y -165.898,Z 57.795,A 37.911,B 90.000,C 0.000} C_DIS
LIN {X -244.883,Y -113.721,Z 168.941,A 24.910,B 90.000,C 0.000} C_DIS
LIN {X -261.208,Y -121.302,Z 168.941,A 24.910,B 90.000,C 0.000} C_DIS
LIN {X -263.022,Y -122.145,Z 168.941,A 24.910,B 90.000,C 0.000} C_DIS
WAIT SEC 1.75
RET=EKI_SetBool("oxy","torchState",TRUE)
RET = EKI_Send("oxy","torchState")
LIN {X -262.392,Y -123.493,Z 170.949,A 25.204,B 90.000,C 0.000} C_DIS
LIN {X -261.826,Y -124.688,Z 173.071,A 25.465,B 90.000,C 0.000} C_DIS
LIN {X -261.320,Y -125.746,Z 175.278,A 25.697,B 90.000,C 0.000} C_DIS
LIN {X -260.862,Y -126.692,Z 177.546,A 25.904,B 90.000,C 0.000} C_DIS
LIN {X -260.444,Y -127.550,Z 179.856,A 26.093,B 90.000,C 0.000} C_DIS
LIN {X -260.052,Y -128.347,Z 182.193,A 26.268,B 90.000,C 0.000} C_DIS
LIN {X -259.674,Y -129.110,Z 184.543,A 26.437,B 90.000,C 0.000} C_DIS
LIN {X -259.409,Y -129.642,Z 186.213,A 26.554,B 90.000,C 0.000} C_DIS
LIN {X -257.620,Y -128.748,Z 186.213,A 26.554,B 90.000,C 0.000} C_DIS
WAIT SEC 0.1
RET=EKI_SetBool("oxy","torchState",FALSE)
RET = EKI_Send("oxy","torchState")
LIN {X -241.518,Y -120.701,Z 186.213,A 26.554,B 90.000,C 0.000} C_DIS
LIN {X -237.649,Y -128.153,Z 203.073,A 28.336,B 90.000,C 0.000} C_DIS
LIN {X -253.492,Y -136.696,Z 203.073,A 28.336,B 90.000,C 0.000} C_DIS
LIN {X -255.252,Y -137.645,Z 203.073,A 28.336,B 90.000,C 0.000} C_DIS
WAIT SEC 1.75
RET=EKI_SetBool("oxy","torchState",TRUE)
RET = EKI_Send("oxy","torchState")
LIN {X -254.380,Y -139.252,Z 204.778,A 28.697,B 90.000,C 0.000} C_DIS
LIN {X -253.418,Y -140.994,Z 206.291,A 29.090,B 90.000,C 0.000} C_DIS
LIN {X -252.378,Y -142.848,Z 207.606,A 29.510,B 90.000,C 0.000} C_DIS
LIN {X -251.270,Y -144.788,Z 208.728,A 29.952,B 90.000,C 0.000} C_DIS
LIN {X -250.104,Y -146.793,Z 209.659,A 30.410,B 90.000,C 0.000} C_DIS
LIN {X -248.887,Y -148.847,Z 210.401,A 30.882,B 90.000,C 0.000} C_DIS
LIN {X -247.628,Y -150.932,Z 210.962,A 31.363,B 90.000,C 0.000} C_DIS
LIN {X -247.251,Y -151.549,Z 211.092,A 31.506,B 90.000,C 0.000} C_DIS
LIN {X -245.545,Y -150.504,Z 211.092,A 31.506,B 90.000,C 0.000} C_DIS
WAIT SEC 0.1
RET=EKI_SetBool("oxy","torchState",FALSE)
RET = EKI_Send("oxy","torchState")
LIN {X -230.199,Y -141.097,Z 211.092,A 31.506,B 90.000,C 0.000} C_DIS
LIN {X -264.659,Y -53.437,Z 241.972,A 11.415,B 90.000,C 0.000} C_DIS
LIN {X -282.303,Y -56.999,Z 241.972,A 11.415,B 90.000,C 0.000} C_DIS
LIN {X -284.264,Y -57.395,Z 241.972,A 11.415,B 90.000,C 0.000} C_DIS
WAIT SEC 1.75
RET=EKI_SetBool("oxy","torchState",TRUE)
RET = EKI_Send("oxy","torchState")
LIN {X -284.526,Y -56.078,Z 239.864,A 11.150,B 90.000,C 0.000} C_DIS
LIN {X -284.794,Y -54.701,Z 237.795,A 10.873,B 90.000,C 0.000} C_DIS
LIN {X -285.066,Y -53.266,Z 235.766,A 10.584,B 90.000,C 0.000} C_DIS
LIN {X -285.341,Y -51.773,Z 233.780,A 10.284,B 90.000,C 0.000} C_DIS
LIN {X -285.618,Y -50.223,Z 231.839,A 9.973,B 90.000,C 0.000} C_DIS
LIN {X -285.895,Y -48.618,Z 229.943,A 9.651,B 90.000,C 0.000} C_DIS
LIN {X -286.172,Y -46.959,Z 228.093,A 9.319,B 90.000,C 0.000} C_DIS
LIN {X -286.448,Y -45.248,Z 226.292,A 8.976,B 90.000,C 0.000} C_DIS
LIN {X -286.721,Y -43.487,Z 224.539,A 8.624,B 90.000,C 0.000} C_DIS
LIN {X -286.989,Y -41.676,Z 222.837,A 8.263,B 90.000,C 0.000} C_DIS
LIN {X -287.253,Y -39.817,Z 221.187,A 7.892,B 90.000,C 0.000} C_DIS
LIN {X -287.511,Y -37.912,Z 219.589,A 7.512,B 90.000,C 0.000} C_DIS
LIN {X -287.761,Y -35.961,Z 218.046,A 7.123,B 90.000,C 0.000} C_DIS
LIN {X -288.004,Y -33.967,Z 216.559,A 6.726,B 90.000,C 0.000} C_DIS
LIN {X -288.237,Y -31.930,Z 215.129,A 6.321,B 90.000,C 0.000} C_DIS
LIN {X -288.459,Y -29.852,Z 213.758,A 5.908,B 90.000,C 0.000} C_DIS
LIN {X -288.670,Y -27.734,Z 212.447,A 5.488,B 90.000,C 0.000} C_DIS
LIN {X -288.869,Y -25.579,Z 211.196,A 5.060,B 90.000,C 0.000} C_DIS
LIN {X -289.055,Y -23.387,Z 210.008,A 4.626,B 90.000,C 0.000} C_DIS
LIN {X -289.226,Y -21.161,Z 208.884,A 4.185,B 90.000,C 0.000} C_DIS
LIN {X -289.330,Y -19.695,Z 208.185,A 3.894,B 90.000,C 0.000} C_DIS
LIN {X -287.335,Y -19.559,Z 208.185,A 3.894,B 90.000,C 0.000} C_DIS
WAIT SEC 0.1
RET=EKI_SetBool("oxy","torchState",FALSE)
RET = EKI_Send("oxy","torchState")
LIN {X -269.377,Y -18.337,Z 208.185,A 3.894,B 90.000,C 0.000} C_DIS
LIN {X -269.998,Y 1.072,Z 166.170,A -0.227,B 90.000,C 0.000} C_DIS
LIN {X -287.998,Y 1.143,Z 166.170,A -0.227,B 90.000,C 0.000} C_DIS
LIN {X -289.998,Y 1.151,Z 166.170,A -0.227,B 90.000,C 0.000} C_DIS
WAIT SEC 1.75
RET=EKI_SetBool("oxy","torchState",TRUE)
RET = EKI_Send("oxy","torchState")
LIN {X -289.977,Y 3.649,Z 166.063,A -0.721,B 90.000,C 0.000} C_DIS
LIN {X -289.935,Y 6.148,Z 166.047,A -1.215,B 90.000,C 0.000} C_DIS
LIN {X -289.871,Y 8.645,Z 166.129,A -1.708,B 90.000,C 0.000} C_DIS
LIN {X -289.786,Y 11.138,Z 166.297,A -2.201,B 90.000,C 0.000} C_DIS
LIN {X -289.680,Y 13.623,Z 166.549,A -2.692,B 90.000,C 0.000} C_DIS
LIN {X -289.553,Y 16.097,Z 166.884,A -3.182,B 90.000,C 0.000} C_DIS
LIN {X -289.405,Y 18.558,Z 167.294,A -3.669,B 90.000,C 0.000} C_DIS
LIN {X -289.238,Y 21.005,Z 167.777,A -4.154,B 90.000,C 0.000} C_DIS
LIN {X -289.051,Y 23.436,Z 168.327,A -4.635,B 90.000,C 0.000} C_DIS
LIN {X -288.845,Y 25.851,Z 168.941,A -5.114,B 90.000,C 0.000} C_DIS
LIN {X -288.620,Y 28.247,Z 169.615,A -5.590,B 90.000,C 0.000} C_DIS
LIN {X -288.378,Y 30.626,Z 170.344,A -6.062,B 90.000,C 0.000} C_DIS
LIN {X -288.118,Y 32.986,Z 171.126,A -6.531,B 90.000,C 0.000} C_DIS
LIN {X -287.840,Y 35.327,Z 171.958,A -6.997,B 90.000,C 0.000} C_DIS
LIN {X -287.545,Y 37.648,Z 172.836,A -7.459,B 90.000,C 0.000} C_DIS
LIN {X -287.456,Y 38.328,Z 173.100,A -7.595,B 90.000,C 0.000} C_DIS
LIN {X -285.474,Y 38.064,Z 173.100,A -7.595,B 90.000,C 0.000} C_DIS
WAIT SEC 0.1
RET=EKI_SetBool("oxy","torchState",FALSE)
RET = EKI_Send("oxy","torchState")
LIN {X -267.631,Y 35.685,Z 173.100,A -7.595,B 90.000,C 0.000} C_DIS
LIN {X -267.654,Y 35.512,Z 202.563,A -7.558,B 90.000,C 0.000} C_DIS
LIN {X -285.498,Y 37.880,Z 202.563,A -7.558,B 90.000,C 0.000} C_DIS
LIN {X -287.481,Y 38.143,Z 202.563,A -7.558,B 90.000,C 0.000} C_DIS
WAIT SEC 1.75
RET=EKI_SetBool("oxy","torchState",TRUE)
RET = EKI_Send("oxy","torchState")
LIN {X -287.152,Y 40.539,Z 203.193,A -8.036,B 90.000,C 0.000} C_DIS
LIN {X -286.807,Y 42.914,Z 203.893,A -8.510,B 90.000,C 0.000} C_DIS
LIN {X -286.445,Y 45.265,Z 204.662,A -8.980,B 90.000,C 0.000} C_DIS
LIN {X -286.068,Y 47.590,Z 205.499,A -9.445,B 90.000,C 0.000} C_DIS
LIN {X -285.676,Y 49.888,Z 206.402,A -9.906,B 90.000,C 0.000} C_DIS
LIN {X -285.271,Y 52.156,Z 207.371,A -10.361,B 90.000,C 0.000} C_DIS
LIN {X -284.853,Y 54.394,Z 208.404,A -10.811,B 90.000,C 0.000} C_DIS
LIN {X -284.423,Y 56.598,Z 209.501,A -11.254,B 90.000,C 0.000} C_DIS
LIN {X -283.983,Y 58.769,Z 210.660,A -11.692,B 90.000,C 0.000} C_DIS
LIN {X -283.533,Y 60.903,Z 211.882,A -12.123,B 90.000,C 0.000} C_DIS
LIN {X -283.074,Y 62.999,Z 213.164,A -12.547,B 90.000,C 0.000} C_DIS
LIN {X -282.608,Y 65.057,Z 214.505,A -12.964,B 90.000,C 0.000} C_DIS
LIN {X -282.136,Y 67.074,Z 215.904,A -13.373,B 90.000,C 0.000} C_DIS
LIN {X -281.659,Y 69.049,Z 217.360,A -13.774,B 90.000,C 0.000} C_DIS
LIN {X -281.179,Y 70.980,Z 218.872,A -14.168,B 90.000,C 0.000} C_DIS
LIN {X -280.696,Y 72.867,Z 220.439,A -14.552,B 90.000,C 0.000} C_DIS
LIN {X -280.212,Y 74.708,Z 222.060,A -14.928,B 90.000,C 0.000} C_DIS
LIN {X -279.728,Y 76.500,Z 223.733,A -15.295,B 90.000,C 0.000} C_DIS
LIN {X -279.245,Y 78.244,Z 225.458,A -15.653,B 90.000,C 0.000} C_DIS
LIN {X -278.766,Y 79.936,Z 227.234,A -16.000,B 90.000,C 0.000} C_DIS
LIN {X -278.290,Y 81.575,Z 229.061,A -16.337,B 90.000,C 0.000} C_DIS
LIN {X -277.820,Y 83.160,Z 230.935,A -16.664,B 90.000,C 0.000} C_DIS
LIN {X -277.358,Y 84.691,Z 232.857,A -16.980,B 90.000,C 0.000} C_DIS
LIN {X -277.023,Y 85.781,Z 234.297,A -17.205,B 90.000,C 0.000} C_DIS
LIN {X -275.112,Y 85.189,Z 234.297,A -17.205,B 90.000,C 0.000} C_DIS
WAIT SEC 0.1
RET=EKI_SetBool("oxy","torchState",FALSE)
RET = EKI_Send("oxy","torchState")
LIN {X -257.918,Y 79.865,Z 234.297,A -17.205,B 90.000,C 0.000} C_DIS
LIN {X -247.232,Y 108.519,Z 209.874,A -23.698,B 90.000,C 0.000} C_DIS
LIN {X -263.714,Y 115.754,Z 209.874,A -23.698,B 90.000,C 0.000} C_DIS
LIN {X -265.545,Y 116.558,Z 209.874,A -23.698,B 90.000,C 0.000} C_DIS
WAIT SEC 1.75
RET=EKI_SetBool("oxy","torchState",TRUE)
RET = EKI_Send("oxy","torchState")
LIN {X -266.481,Y 114.402,Z 209.021,A -23.234,B 90.000,C 0.000} C_DIS
LIN {X -267.397,Y 112.245,Z 208.152,A -22.771,B 90.000,C 0.000} C_DIS
LIN {X -268.293,Y 110.084,Z 207.270,A -22.309,B 90.000,C 0.000} C_DIS
LIN {X -269.170,Y 107.922,Z 206.373,A -21.848,B 90.000,C 0.000} C_DIS
LIN {X -270.027,Y 105.758,Z 205.462,A -21.388,B 90.000,C 0.000} C_DIS
LIN {X -270.865,Y 103.592,Z 204.538,A -20.929,B 90.000,C 0.000} C_DIS
LIN {X -271.684,Y 101.425,Z 203.599,A -20.472,B 90.000,C 0.000} C_DIS
LIN {X -272.483,Y 99.256,Z 202.647,A -20.015,B 90.000,C 0.000} C_DIS
LIN {X -273.264,Y 97.086,Z 201.681,A -19.559,B 90.000,C 0.000} C_DIS
LIN {X -274.025,Y 94.916,Z 200.702,A -19.105,B 90.000,C 0.000} C_DIS
LIN {X -274.767,Y 92.745,Z 199.710,A -18.652,B 90.000,C 0.000} C_DIS
LIN {X -275.490,Y 90.574,Z 198.704,A -18.199,B 90.000,C 0.000} C_DIS
LIN {X -276.195,Y 88.403,Z 197.686,A -17.748,B 90.000,C 0.000} C_DIS
LIN {X -276.880,Y 86.231,Z 196.654,A -17.299,B 90.000,C 0.000} C_DIS
LIN {X -277.547,Y 84.060,Z 195.610,A -16.850,B 90.000,C 0.000} C_DIS
LIN {X -278.195,Y 81.890,Z 194.553,A -16.402,B 90.000,C 0.000} C_DIS
LIN {X -278.825,Y 79.720,Z 193.484,A -15.956,B 90.000,C 0.000} C_DIS
LIN {X -279.437,Y 77.551,Z 192.402,A -15.511,B 90.000,C 0.000} C_DIS
LIN {X -280.030,Y 75.383,Z 191.308,A -15.067,B 90.000,C 0.000} C_DIS
LIN {X -280.605,Y 73.217,Z 190.201,A -14.624,B 90.000,C 0.000} C_DIS
LIN {X -280.887,Y 72.129,Z 189.641,A -14.402,B 90.000,C 0.000} C_DIS
LIN {X -278.950,Y 71.632,Z 189.641,A -14.402,B 90.000,C 0.000} C_DIS
WAIT SEC 0.1
RET=EKI_SetBool("oxy","torchState",FALSE)
RET = EKI_Send("oxy","torchState")
LIN {X -261.515,Y 67.155,Z 189.641,A -14.402,B 90.000,C 0.000} C_DIS
LIN {X -259.856,Y 73.314,Z 148.655,A -15.756,B 90.000,C 0.000} C_DIS
LIN {X -277.179,Y 78.202,Z 148.655,A -15.756,B 90.000,C 0.000} C_DIS
LIN {X -279.104,Y 78.745,Z 148.655,A -15.756,B 90.000,C 0.000} C_DIS
WAIT SEC 1.75
RET=EKI_SetBool("oxy","torchState",TRUE)
RET = EKI_Send("oxy","torchState")
LIN {X -279.631,Y 76.853,Z 147.109,A -15.367,B 90.000,C 0.000} C_DIS
LIN {X -280.156,Y 74.919,Z 145.614,A -14.972,B 90.000,C 0.000} C_DIS
LIN {X -280.677,Y 72.942,Z 144.177,A -14.568,B 90.000,C 0.000} C_DIS
LIN {X -281.194,Y 70.919,Z 142.802,A -14.155,B 90.000,C 0.000} C_DIS
LIN {X -281.708,Y 68.851,Z 141.496,A -13.734,B 90.000,C 0.000} C_DIS
LIN {X -282.217,Y 66.736,Z 140.264,A -13.304,B 90.000,C 0.000} C_DIS
LIN {X -282.719,Y 64.572,Z 139.118,A -12.865,B 90.000,C 0.000} C_DIS
LIN {X -283.215,Y 62.362,Z 138.061,A -12.418,B 90.000,C 0.000} C_DIS
LIN {X -283.703,Y 60.103,Z 137.107,A -11.961,B 90.000,C 0.000} C_DIS
LIN {X -284.181,Y 57.800,Z 136.261,A -11.497,B 90.000,C 0.000} C_DIS
LIN {X -284.648,Y 55.455,Z 135.533,A -11.024,B 90.000,C 0.000} C_DIS
LIN {X -285.102,Y 53.071,Z 134.932,A -10.545,B 90.000,C 0.000} C_DIS
LIN {X -285.542,Y 50.655,Z 134.467,A -10.060,B 90.000,C 0.000} C_DIS
LIN {X -285.668,Y 49.940,Z 134.358,A -9.916,B 90.000,C 0.000} C_DIS
LIN {X -283.697,Y 49.596,Z 134.358,A -9.916,B 90.000,C 0.000} C_DIS
WAIT SEC 0.1
RET=EKI_SetBool("oxy","torchState",FALSE)
RET = EKI_Send("oxy","torchState")
LIN {X -265.966,Y 46.496,Z 134.358,A -9.916,B 90.000,C 0.000} C_DIS
LIN {X -236.508,Y 130.247,Z 199.192,A -28.842,B 90.000,C 0.000} C_DIS
LIN {X -252.275,Y 138.930,Z 199.192,A -28.842,B 90.000,C 0.000} C_DIS
LIN {X -254.027,Y 139.895,Z 199.192,A -28.842,B 90.000,C 0.000} C_DIS
WAIT SEC 1.75
RET=EKI_SetBool("oxy","torchState",TRUE)
RET = EKI_Send("oxy","torchState")
LIN {X -252.924,Y 141.877,Z 200.241,A -29.290,B 90.000,C 0.000} C_DIS
LIN {X -251.798,Y 143.865,Z 201.257,A -29.741,B 90.000,C 0.000} C_DIS
LIN {X -250.651,Y 145.856,Z 202.239,A -30.196,B 90.000,C 0.000} C_DIS
LIN {X -249.478,Y 147.851,Z 203.185,A -30.653,B 90.000,C 0.000} C_DIS
LIN {X -248.285,Y 149.849,Z 204.098,A -31.112,B 90.000,C 0.000} C_DIS
LIN {X -247.066,Y 151.848,Z 204.973,A -31.575,B 90.000,C 0.000} C_DIS
LIN {X -245.826,Y 153.849,Z 205.814,A -32.040,B 90.000,C 0.000} C_DIS
LIN {X -244.561,Y 155.850,Z 206.617,A -32.508,B 90.000,C 0.000} C_DIS
LIN {X -243.275,Y 157.851,Z 207.384,A -32.978,B 90.000,C 0.000} C_DIS
LIN {X -241.965,Y 159.852,Z 208.113,A -33.450,B 90.000,C 0.000} C_DIS
LIN {X -240.632,Y 161.850,Z 208.805,A -33.925,B 90.000,C 0.000} C_DIS
LIN {X -239.278,Y 163.847,Z 209.460,A -34.402,B 90.000,C 0.000} C_DIS
LIN {X -237.900,Y 165.840,Z 210.074,A -34.880,B 90.000,C 0.000} C_DIS
LIN {X -236.502,Y 167.829,Z 210.652,A -35.361,B 90.000,C 0.000} C_DIS
LIN {X -235.080,Y 169.814,Z 211.188,A -35.843,B 90.000,C 0.000} C_DIS
LIN {X -233.637,Y 171.794,Z 211.687,A -36.327,B 90.000,C 0.000} C_DIS
LIN {X -232.173,Y 173.768,Z 212.145,A -36.813,B 90.000,C 0.000} C_DIS
LIN {X -230.688,Y 175.734,Z 212.561,A -37.300,B 90.000,C 0.000} C_DIS
LIN {X -229.183,Y 177.694,Z 212.940,A -37.788,B 90.000,C 0.000} C_DIS
LIN {X -227.656,Y 179.645,Z 213.274,A -38.277,B 90.000,C 0.000} C_DIS
LIN {X -227.335,Y 180.052,Z 213.341,A -38.380,B 90.000,C 0.000} C_DIS
LIN {X -225.767,Y 178.810,Z 213.341,A -38.380,B 90.000,C 0.000} C_DIS
WAIT SEC 0.1
RET=EKI_SetBool("oxy","torchState",FALSE)
RET = EKI_Send("oxy","torchState")
LIN {X -211.657,Y 167.635,Z 213.341,A -38.380,B 90.000,C 0.000} C_DIS
LIN {X -225.344,Y 148.728,Z 223.979,A -33.425,B 90.000,C 0.000} C_DIS
LIN {X -240.367,Y 158.643,Z 223.979,A -33.425,B 90.000,C 0.000} C_DIS
LIN {X -242.037,Y 159.744,Z 223.979,A -33.425,B 90.000,C 0.000} C_DIS
WAIT SEC 1.75
RET=EKI_SetBool("oxy","torchState",TRUE)
RET = EKI_Send("oxy","torchState")
LIN {X -240.678,Y 161.780,Z 224.489,A -33.908,B 90.000,C 0.000} C_DIS
LIN {X -239.303,Y 163.808,Z 224.981,A -34.393,B 90.000,C 0.000} C_DIS
LIN {X -237.909,Y 165.828,Z 225.455,A -34.877,B 90.000,C 0.000} C_DIS
LIN {X -236.495,Y 167.839,Z 225.909,A -35.363,B 90.000,C 0.000} C_DIS
LIN {X -235.061,Y 169.840,Z 226.342,A -35.850,B 90.000,C 0.000} C_DIS
LIN {X -233.608,Y 171.832,Z 226.754,A -36.337,B 90.000,C 0.000} C_DIS
LIN {X -232.136,Y 173.815,Z 227.145,A -36.824,B 90.000,C 0.000} C_DIS
LIN {X -230.646,Y 175.788,Z 227.516,A -37.313,B 90.000,C 0.000} C_DIS
LIN {X -229.138,Y 177.750,Z 227.865,A -37.802,B 90.000,C 0.000} C_DIS
LIN {X -227.611,Y 179.702,Z 228.191,A -38.292,B 90.000,C 0.000} C_DIS
LIN {X -226.064,Y 181.643,Z 228.492,A -38.782,B 90.000,C 0.000} C_DIS
LIN {X -224.500,Y 183.572,Z 228.771,A -39.273,B 90.000,C 0.000} C_DIS
LIN {X -222.918,Y 185.491,Z 229.026,A -39.764,B 90.000,C 0.000} C_DIS
LIN {X -221.319,Y 187.398,Z 229.257,A -40.256,B 90.000,C 0.000} C_DIS
LIN {X -219.700,Y 189.292,Z 229.460,A -40.748,B 90.000,C 0.000} C_DIS
LIN {X -218.064,Y 191.173,Z 229.638,A -41.241,B 90.000,C 0.000} C_DIS
LIN {X -216.412,Y 193.043,Z 229.791,A -41.734,B 90.000,C 0.000} C_DIS
LIN {X -214.742,Y 194.899,Z 229.916,A -42.227,B 90.000,C 0.000} C_DIS
LIN {X -213.055,Y 196.741,Z 230.012,A -42.720,B 90.000,C 0.000} C_DIS
LIN {X -211.352,Y 198.570,Z 230.082,A -43.214,B 90.000,C 0.000} C_DIS
LIN {X -209.633,Y 200.384,Z 230.122,A -43.708,B 90.000,C 0.000} C_DIS
LIN {X -208.652,Y 201.406,Z 230.133,A -43.988,B 90.000,C 0.000} C_DIS
LIN {X -207.213,Y 200.017,Z 230.133,A -43.988,B 90.000,C 0.000} C_DIS
WAIT SEC 0.1
RET=EKI_SetBool("oxy","torchState",FALSE)
RET = EKI_Send("oxy","torchState")
LIN {X -194.262,Y 187.516,Z 230.133,A -43.988,B 90.000,C 0.000} C_DIS
LIN {X -185.001,Y 196.658,Z 213.259,A -46.749,B 90.000,C 0.000} C_DIS
LIN {X -197.335,Y 209.769,Z 213.259,A -46.749,B 90.000,C 0.000} C_DIS
LIN {X -198.705,Y 211.225,Z 213.259,A -46.749,B 90.000,C 0.000} C_DIS
WAIT SEC 1.75
RET=EKI_SetBool("oxy","torchState",TRUE)
RET = EKI_Send("oxy","torchState")
LIN {X -196.889,Y 212.917,Z 212.963,A -47.240,B 90.000,C 0.000} C_DIS
LIN {X -195.062,Y 214.593,Z 212.644,A -47.730,B 90.000,C 0.000} C_DIS
LIN {X -193.223,Y 216.251,Z 212.297,A -48.219,B 90.000,C 0.000} C_DIS
LIN {X -191.373,Y 217.889,Z 211.924,A -48.707,B 90.000,C 0.000} C_DIS
LIN {X -189.511,Y 219.510,Z 211.527,A -49.195,B 90.000,C 0.000} C_DIS
LIN {X -187.640,Y 221.113,Z 211.107,A -49.681,B 90.000,C 0.000} C_DIS
LIN {X -185.758,Y 222.697,Z 210.663,A -50.168,B 90.000,C 0.000} C_DIS
LIN {X -183.865,Y 224.261,Z 210.195,A -50.653,B 90.000,C 0.000} C_DIS
LIN {X -181.962,Y 225.807,Z 209.706,A -51.137,B 90.000,C 0.000} C_DIS
LIN {X -180.050,Y 227.334,Z 209.196,A -51.621,B 90.000,C 0.000} C_DIS
LIN {X -178.129,Y 228.843,Z 208.666,A -52.103,B 90.000,C 0.000} C_DIS
LIN {X -176.199,Y 230.333,Z 208.117,A -52.585,B 90.000,C 0.000} C_DIS
LIN {X -174.259,Y 231.804,Z 207.548,A -53.066,B 90.000,C 0.000} C_DIS
LIN {X -172.311,Y 233.256,Z 206.961,A -53.546,B 90.000,C 0.000} C_DIS
LIN {X -170.354,Y 234.690,Z 206.357,A -54.025,B 90.000,C 0.000} C_DIS
LIN {X -168.389,Y 236.104,Z 205.735,A -54.504,B 90.000,C 0.000} C_DIS
LIN {X -166.443,Y 237.480,Z 205.106,A -54.974,B 90.000,C 0.000} C_DIS
LIN {X -165.295,Y 235.842,Z 205.106,A -54.974,B 90.000,C 0.000} C_DIS
WAIT SEC 0.1
RET=EKI_SetBool("oxy","torchState",FALSE)
RET = EKI_Send("oxy","torchState")
LIN {X -154.964,Y 221.102,Z 205.106,A -54.974,B 90.000,C 0.000} C_DIS
LIN {X -156.859,Y 219.762,Z 222.344,A -54.482,B 90.000,C 0.000} C_DIS
LIN {X -167.316,Y 234.413,Z 222.344,A -54.482,B 90.000,C 0.000} C_DIS
LIN {X -168.478,Y 236.040,Z 222.344,A -54.482,B 90.000,C 0.000} C_DIS
WAIT SEC 1.75
RET=EKI_SetBool("oxy","torchState",TRUE)
RET = EKI_Send("oxy","torchState")
LIN {X -166.543,Y 237.410,Z 221.552,A -54.950,B 90.000,C 0.000} C_DIS
LIN {X -164.606,Y 238.757,Z 220.727,A -55.417,B 90.000,C 0.000} C_DIS
LIN {X -162.665,Y 240.083,Z 219.875,A -55.881,B 90.000,C 0.000} C_DIS
LIN {X -160.720,Y 241.388,Z 219.003,A -56.344,B 90.000,C 0.000} C_DIS
LIN {X -158.767,Y 242.675,Z 218.120,A -56.806,B 90.000,C 0.000} C_DIS
LIN {X -156.806,Y 243.947,Z 217.234,A -57.268,B 90.000,C 0.000} C_DIS
LIN {X -154.837,Y 245.205,Z 216.347,A -57.729,B 90.000,C 0.000} C_DIS
LIN {X -152.852,Y 246.447,Z 215.470,A -58.192,B 90.000,C 0.000} C_DIS
LIN {X -150.852,Y 247.675,Z 214.611,A -58.656,B 90.000,C 0.000} C_DIS
LIN {X -148.836,Y 248.892,Z 213.773,A -59.121,B 90.000,C 0.000} C_DIS
LIN {X -146.800,Y 250.099,Z 212.967,A -59.588,B 90.000,C 0.000} C_DIS
LIN {X -144.745,Y 251.294,Z 212.197,A -60.058,B 90.000,C 0.000} C_DIS
LIN {X -143.540,Y 251.984,Z 211.770,A -60.332,B 90.000,C 0.000} C_DIS
LIN {X -142.550,Y 250.247,Z 211.770,A -60.332,B 90.000,C 0.000} C_DIS
WAIT SEC 0.1
RET=EKI_SetBool("oxy","torchState",FALSE)
RET = EKI_Send("oxy","torchState")
LIN {X -133.641,Y 234.606,Z 211.770,A -60.332,B 90.000,C 0.000} C_DIS
LIN {X -132.283,Y 235.374,Z 199.231,A -60.663,B 90.000,C 0.000} C_DIS
LIN {X -141.102,Y 251.066,Z 199.231,A -60.663,B 90.000,C 0.000} C_DIS
LIN {X -142.082,Y 252.810,Z 199.231,A -60.663,B 90.000,C 0.000} C_DIS
WAIT SEC 1.75
RET=EKI_SetBool("oxy","torchState",TRUE)
RET = EKI_Send("oxy","torchState")
LIN {X -139.898,Y 254.024,Z 199.168,A -61.157,B 90.000,C 0.000} C_DIS
LIN {X -137.703,Y 255.220,Z 199.155,A -61.651,B 90.000,C 0.000} C_DIS
LIN {X -135.498,Y 256.398,Z 199.142,A -62.145,B 90.000,C 0.000} C_DIS
LIN {X -133.284,Y 257.556,Z 199.071,A -62.639,B 90.000,C 0.000} C_DIS
LIN {X -131.065,Y 258.693,Z 198.891,A -63.131,B 90.000,C 0.000} C_DIS
LIN {X -128.852,Y 259.802,Z 198.545,A -63.620,B 90.000,C 0.000} C_DIS
LIN {X -126.661,Y 260.877,Z 198.006,A -64.103,B 90.000,C 0.000} C_DIS
LIN {X -124.501,Y 261.915,Z 197.293,A -64.576,B 90.000,C 0.000} C_DIS
LIN {X -122.378,Y 262.914,Z 196.432,A -65.040,B 90.000,C 0.000} C_DIS
LIN {X -120.291,Y 263.875,Z 195.447,A -65.494,B 90.000,C 0.000} C_DIS
LIN {X -118.236,Y 264.802,Z 194.367,A -65.939,B 90.000,C 0.000} C_DIS
LIN {X -116.209,Y 265.698,Z 193.211,A -66.377,B 90.000,C 0.000} C_DIS
LIN {X -114.202,Y 266.567,Z 192.000,A -66.809,B 90.000,C 0.000} C_DIS
LIN {X -113.236,Y 266.979,Z 191.401,A -67.016,B 90.000,C 0.000} C_DIS
LIN {X -112.455,Y 265.137,Z 191.401,A -67.016,B 90.000,C 0.000} C_DIS
WAIT SEC 0.1
RET=EKI_SetBool("oxy","torchState",FALSE)
RET = EKI_Send("oxy","torchState")
LIN {X -105.427,Y 248.566,Z 191.401,A -67.016,B 90.000,C 0.000} C_DIS
LIN {X -90.520,Y 254.374,Z 182.654,A -70.412,B 90.000,C 0.000} C_DIS
LIN {X -96.555,Y 271.332,Z 182.654,A -70.412,B 90.000,C 0.000} C_DIS
LIN {X -97.226,Y 273.216,Z 182.654,A -70.412,B 90.000,C 0.000} C_DIS
WAIT SEC 1.75
RET=EKI_SetBool("oxy","torchState",TRUE)
RET = EKI_Send("oxy","torchState")
LIN {X -94.969,Y 274.009,Z 181.926,A -70.884,B 90.000,C 0.000} C_DIS
LIN {X -92.670,Y 274.795,Z 181.339,A -71.364,B 90.000,C 0.000} C_DIS
LIN {X -90.337,Y 275.571,Z 180.891,A -71.850,B 90.000,C 0.000} C_DIS
LIN {X -87.977,Y 276.333,Z 180.576,A -72.340,B 90.000,C 0.000} C_DIS
LIN {X -85.599,Y 277.079,Z 180.386,A -72.832,B 90.000,C 0.000} C_DIS
LIN {X -83.208,Y 277.806,Z 180.318,A -73.326,B 90.000,C 0.000} C_DIS
LIN {X -80.811,Y 278.513,Z 180.360,A -73.820,B 90.000,C 0.000} C_DIS
LIN {X -78.411,Y 279.198,Z 180.506,A -74.313,B 90.000,C 0.000} C_DIS
LIN {X -76.013,Y 279.860,Z 180.747,A -74.804,B 90.000,C 0.000} C_DIS
LIN {X -73.619,Y 280.499,Z 181.077,A -75.294,B 90.000,C 0.000} C_DIS
LIN {X -71.231,Y 281.115,Z 181.487,A -75.781,B 90.000,C 0.000} C_DIS
LIN {X -68.852,Y 281.708,Z 181.972,A -76.266,B 90.000,C 0.000} C_DIS
LIN {X -66.481,Y 282.276,Z 182.525,A -76.747,B 90.000,C 0.000} C_DIS
LIN {X -64.121,Y 282.822,Z 183.142,A -77.226,B 90.000,C 0.000} C_DIS
LIN {X -61.771,Y 283.344,Z 183.815,A -77.702,B 90.000,C 0.000} C_DIS
LIN {X -59.929,Y 283.740,Z 184.379,A -78.074,B 90.000,C 0.000} C_DIS
LIN {X -59.516,Y 281.783,Z 184.379,A -78.074,B 90.000,C 0.000} C_DIS
WAIT SEC 0.1
RET=EKI_SetBool("oxy","torchState",FALSE)
RET = EKI_Send("oxy","torchState")
LIN {X -55.796,Y 264.172,Z 184.379,A -78.074,B 90.000,C 0.000} C_DIS
LIN {X -43.538,Y 266.467,Z 152.644,A -80.721,B 90.000,C 0.000} C_DIS
LIN {X -46.440,Y 284.231,Z 152.644,A -80.721,B 90.000,C 0.000} C_DIS
LIN {X -46.763,Y 286.205,Z 152.644,A -80.721,B 90.000,C 0.000} C_DIS
WAIT SEC 1.75
RET=EKI_SetBool("oxy","torchState",TRUE)
RET = EKI_Send("oxy","torchState")
LIN {X -49.115,Y 285.810,Z 151.895,A -80.249,B 90.000,C 0.000} C_DIS
LIN {X -51.474,Y 285.395,Z 151.181,A -79.776,B 90.000,C 0.000} C_DIS
LIN {X -53.841,Y 284.957,Z 150.508,A -79.300,B 90.000,C 0.000} C_DIS
LIN {X -56.215,Y 284.498,Z 149.872,A -78.823,B 90.000,C 0.000} C_DIS
LIN {X -58.594,Y 284.019,Z 149.275,A -78.343,B 90.000,C 0.000} C_DIS
LIN {X -60.979,Y 283.515,Z 148.718,A -77.862,B 90.000,C 0.000} C_DIS
LIN {X -63.367,Y 282.992,Z 148.199,A -77.379,B 90.000,C 0.000} C_DIS
LIN {X -65.759,Y 282.445,Z 147.722,A -76.894,B 90.000,C 0.000} C_DIS
LIN {X -68.154,Y 281.877,Z 147.284,A -76.408,B 90.000,C 0.000} C_DIS
LIN {X -69.910,Y 281.447,Z 146.987,A -76.050,B 90.000,C 0.000} C_DIS
LIN {X -69.428,Y 279.506,Z 146.987,A -76.050,B 90.000,C 0.000} C_DIS
WAIT SEC 0.1
RET=EKI_SetBool("oxy","torchState",FALSE)
RET = EKI_Send("oxy","torchState")
LIN {X -65.089,Y 262.037,Z 146.987,A -76.050,B 90.000,C 0.000} C_DIS
LIN {X -52.463,Y 264.854,Z 131.908,A -78.796,B 90.000,C 0.000} C_DIS
LIN {X -55.961,Y 282.511,Z 131.908,A -78.796,B 90.000,C 0.000} C_DIS
LIN {X -56.349,Y 284.473,Z 131.908,A -78.796,B 90.000,C 0.000} C_DIS
WAIT SEC 1.75
RET=EKI_SetBool("oxy","torchState",TRUE)
RET = EKI_Send("oxy","torchState")
LIN {X -53.945,Y 284.933,Z 132.411,A -79.279,B 90.000,C 0.000} C_DIS
LIN {X -51.537,Y 285.380,Z 132.916,A -79.763,B 90.000,C 0.000} C_DIS
LIN {X -49.127,Y 285.806,Z 133.424,A -80.247,B 90.000,C 0.000} C_DIS
LIN {X -46.714,Y 286.212,Z 133.932,A -80.730,B 90.000,C 0.000} C_DIS
LIN {X -44.297,Y 286.593,Z 134.445,A -81.214,B 90.000,C 0.000} C_DIS
LIN {X -41.878,Y 286.956,Z 134.959,A -81.697,B 90.000,C 0.000} C_DIS
LIN {X -39.456,Y 287.300,Z 135.474,A -82.180,B 90.000,C 0.000} C_DIS
LIN {X -37.033,Y 287.625,Z 135.994,A -82.663,B 90.000,C 0.000} C_DIS
LIN {X -34.606,Y 287.925,Z 136.514,A -83.146,B 90.000,C 0.000} C_DIS
LIN {X -32.178,Y 288.205,Z 137.038,A -83.629,B 90.000,C 0.000} C_DIS
LIN {X -29.748,Y 288.466,Z 137.564,A -84.112,B 90.000,C 0.000} C_DIS
LIN {X -27.317,Y 288.709,Z 138.091,A -84.595,B 90.000,C 0.000} C_DIS
LIN {X -24.884,Y 288.929,Z 138.622,A -85.077,B 90.000,C 0.000} C_DIS
LIN {X -22.450,Y 289.126,Z 139.154,A -85.560,B 90.000,C 0.000} C_DIS
LIN {X -20.015,Y 289.304,Z 139.689,A -86.042,B 90.000,C 0.000} C_DIS
LIN {X -17.579,Y 289.464,Z 140.227,A -86.525,B 90.000,C 0.000} C_DIS
LIN {X -15.141,Y 289.604,Z 140.765,A -87.007,B 90.000,C 0.000} C_DIS
LIN {X -15.025,Y 289.610,Z 140.791,A -87.030,B 90.000,C 0.000} C_DIS
LIN {X -14.922,Y 287.613,Z 140.791,A -87.030,B 90.000,C 0.000} C_DIS
WAIT SEC 0.1
RET=EKI_SetBool("oxy","torchState",FALSE)
RET = EKI_Send("oxy","torchState")
LIN {X -13.989,Y 269.637,Z 140.791,A -87.030,B 90.000,C 0.000} C_DIS
LIN {X -7.544,Y 269.895,Z 122.911,A -88.399,B 90.000,C 0.000} C_DIS
LIN {X -8.047,Y 287.888,Z 122.911,A -88.399,B 90.000,C 0.000} C_DIS
LIN {X -8.103,Y 289.887,Z 122.911,A -88.399,B 90.000,C 0.000} C_DIS
WAIT SEC 1.75
RET=EKI_SetBool("oxy","torchState",TRUE)
RET = EKI_Send("oxy","torchState")
LIN {X -10.531,Y 289.805,Z 122.322,A -87.919,B 90.000,C 0.000} C_DIS
LIN {X -12.956,Y 289.706,Z 121.726,A -87.439,B 90.000,C 0.000} C_DIS
LIN {X -15.379,Y 289.589,Z 121.122,A -86.960,B 90.000,C 0.000} C_DIS
LIN {X -17.799,Y 289.452,Z 120.510,A -86.481,B 90.000,C 0.000} C_DIS
LIN {X -20.215,Y 289.290,Z 119.889,A -86.003,B 90.000,C 0.000} C_DIS
LIN {X -22.627,Y 289.111,Z 119.260,A -85.525,B 90.000,C 0.000} C_DIS
LIN {X -25.037,Y 288.916,Z 118.624,A -85.047,B 90.000,C 0.000} C_DIS
LIN {X -27.442,Y 288.696,Z 117.978,A -84.570,B 90.000,C 0.000} C_DIS
LIN {X -29.842,Y 288.456,Z 117.324,A -84.093,B 90.000,C 0.000} C_DIS
LIN {X -32.239,Y 288.199,Z 116.663,A -83.617,B 90.000,C 0.000} C_DIS
LIN {X -34.632,Y 287.925,Z 115.995,A -83.141,B 90.000,C 0.000} C_DIS
LIN {X -37.019,Y 287.624,Z 115.315,A -82.666,B 90.000,C 0.000} C_DIS
LIN {X -39.402,Y 287.306,Z 114.629,A -82.191,B 90.000,C 0.000} C_DIS
LIN {X -41.780,Y 286.972,Z 113.935,A -81.717,B 90.000,C 0.000} C_DIS
LIN {X -44.153,Y 286.618,Z 113.234,A -81.243,B 90.000,C 0.000} C_DIS
LIN {X -46.519,Y 286.240,Z 112.522,A -80.769,B 90.000,C 0.000} C_DIS
LIN {X -48.881,Y 285.846,Z 111.803,A -80.296,B 90.000,C 0.000} C_DIS
LIN {X -51.237,Y 285.436,Z 111.078,A -79.823,B 90.000,C 0.000} C_DIS
LIN {X -53.587,Y 285.003,Z 110.342,A -79.351,B 90.000,C 0.000} C_DIS
LIN {X -55.930,Y 284.551,Z 109.599,A -78.880,B 90.000,C 0.000} C_DIS
LIN {X -58.268,Y 284.082,Z 108.848,A -78.409,B 90.000,C 0.000} C_DIS
LIN {X -60.600,Y 283.597,Z 108.090,A -77.938,B 90.000,C 0.000} C_DIS
LIN {X -62.924,Y 283.088,Z 107.322,A -77.468,B 90.000,C 0.000} C_DIS
LIN {X -65.241,Y 282.561,Z 106.546,A -76.999,B 90.000,C 0.000} C_DIS
LIN {X -67.552,Y 282.020,Z 105.764,A -76.530,B 90.000,C 0.000} C_DIS
LIN {X -69.857,Y 281.459,Z 104.973,A -76.061,B 90.000,C 0.000} C_DIS
LIN {X -72.152,Y 280.877,Z 104.173,A -75.593,B 90.000,C 0.000} C_DIS
LIN {X -74.441,Y 280.279,Z 103.365,A -75.126,B 90.000,C 0.000} C_DIS
LIN {X -76.136,Y 279.827,Z 102.763,A -74.779,B 90.000,C 0.000} C_DIS
LIN {X -75.611,Y 277.897,Z 102.763,A -74.779,B 90.000,C 0.000} C_DIS
WAIT SEC 0.1
RET=EKI_SetBool("oxy","torchState",FALSE)
RET = EKI_Send("oxy","torchState")
LIN {X -70.885,Y 260.529,Z 102.763,A -74.779,B 90.000,C 0.000} C_DIS
LIN {X -75.891,Y 259.115,Z 126.357,A -73.676,B 90.000,C 0.000} C_DIS
LIN {X -80.950,Y 276.389,Z 126.357,A -73.676,B 90.000,C 0.000} C_DIS
LIN {X -81.512,Y 278.309,Z 126.357,A -73.676,B 90.000,C 0.000} C_DIS
WAIT SEC 1.75
RET=EKI_SetBool("oxy","torchState",TRUE)
RET = EKI_Send("oxy","torchState")
LIN {X -83.840,Y 277.616,Z 125.765,A -73.196,B 90.000,C 0.000} C_DIS
LIN {X -86.156,Y 276.905,Z 125.150,A -72.717,B 90.000,C 0.000} C_DIS
LIN {X -88.460,Y 276.178,Z 124.510,A -72.240,B 90.000,C 0.000} C_DIS
LIN {X -90.751,Y 275.434,Z 123.840,A -71.764,B 90.000,C 0.000} C_DIS
LIN {X -93.025,Y 274.674,Z 123.133,A -71.290,B 90.000,C 0.000} C_DIS
LIN {X -95.282,Y 273.900,Z 122.389,A -70.819,B 90.000,C 0.000} C_DIS
LIN {X -97.520,Y 273.111,Z 121.602,A -70.350,B 90.000,C 0.000} C_DIS
LIN {X -99.735,Y 272.310,Z 120.767,A -69.884,B 90.000,C 0.000} C_DIS
LIN {X -101.927,Y 271.497,Z 119.881,A -69.423,B 90.000,C 0.000} C_DIS
LIN {X -104.092,Y 270.674,Z 118.941,A -68.965,B 90.000,C 0.000} C_DIS
LIN {X -106.228,Y 269.843,Z 117.942,A -68.512,B 90.000,C 0.000} C_DIS
LIN {X -108.330,Y 269.006,Z 116.881,A -68.065,B 90.000,C 0.000} C_DIS
LIN {X -110.397,Y 268.165,Z 115.754,A -67.624,B 90.000,C 0.000} C_DIS
LIN {X -112.423,Y 267.322,Z 114.557,A -67.191,B 90.000,C 0.000} C_DIS
LIN {X -114.404,Y 266.480,Z 113.286,A -66.765,B 90.000,C 0.000} C_DIS
LIN {X -116.336,Y 265.642,Z 111.940,A -66.349,B 90.000,C 0.000} C_DIS
LIN {X -118.217,Y 264.811,Z 110.518,A -65.943,B 90.000,C 0.000} C_DIS
LIN {X -119.559,Y 264.208,Z 109.424,A -65.652,B 90.000,C 0.000} C_DIS
LIN {X -118.735,Y 262.385,Z 109.424,A -65.652,B 90.000,C 0.000} C_DIS
WAIT SEC 0.1
RET=EKI_SetBool("oxy","torchState",FALSE)
RET = EKI_Send("oxy","torchState")
LIN {X -111.314,Y 245.986,Z 109.424,A -65.652,B 90.000,C 0.000} C_DIS
LIN {X -127.373,Y 238.067,Z 94.713,A -61.852,B 90.000,C 0.000} C_DIS
LIN {X -135.865,Y 253.938,Z 94.713,A -61.852,B 90.000,C 0.000} C_DIS
LIN {X -136.809,Y 255.702,Z 94.713,A -61.852,B 90.000,C 0.000} C_DIS
WAIT SEC 1.75
RET=EKI_SetBool("oxy","torchState",TRUE)
RET = EKI_Send("oxy","torchState")
LIN {X -138.797,Y 254.628,Z 93.644,A -61.405,B 90.000,C 0.000} C_DIS
LIN {X -140.704,Y 253.579,Z 92.415,A -60.975,B 90.000,C 0.000} C_DIS
LIN {X -142.344,Y 252.662,Z 90.767,A -60.604,B 90.000,C 0.000} C_DIS
LIN {X -143.858,Y 251.804,Z 88.972,A -60.260,B 90.000,C 0.000} C_DIS
LIN {X -144.518,Y 251.425,Z 88.329,A -60.110,B 90.000,C 0.000} C_DIS
LIN {X -143.521,Y 249.691,Z 88.329,A -60.110,B 90.000,C 0.000} C_DIS
WAIT SEC 0.1
RET=EKI_SetBool("oxy","torchState",FALSE)
RET = EKI_Send("oxy","torchState")
LIN {X -134.551,Y 234.085,Z 88.329,A -60.110,B 90.000,C 0.000} C_DIS
LIN {X -140.756,Y 230.408,Z 104.428,A -58.579,B 90.000,C 0.000} C_DIS
LIN {X -150.140,Y 245.768,Z 104.428,A -58.579,B 90.000,C 0.000} C_DIS
LIN {X -151.183,Y 247.475,Z 104.428,A -58.579,B 90.000,C 0.000} C_DIS
WAIT SEC 1.75
RET=EKI_SetBool("oxy","torchState",TRUE)
RET = EKI_Send("oxy","torchState")
LIN {X -150.950,Y 247.617,Z 106.913,A -58.633,B 90.000,C 0.000} C_DIS
LIN {X -150.874,Y 247.663,Z 109.411,A -58.651,B 90.000,C 0.000} C_DIS
LIN {X -150.947,Y 247.619,Z 111.909,A -58.634,B 90.000,C 0.000} C_DIS
LIN {X -151.157,Y 247.491,Z 114.397,A -58.585,B 90.000,C 0.000} C_DIS
LIN {X -151.487,Y 247.289,Z 116.866,A -58.509,B 90.000,C 0.000} C_DIS
LIN {X -151.925,Y 247.020,Z 119.313,A -58.407,B 90.000,C 0.000} C_DIS
LIN {X -152.459,Y 246.691,Z 121.733,A -58.283,B 90.000,C 0.000} C_DIS
LIN {X -153.071,Y 246.311,Z 124.126,A -58.141,B 90.000,C 0.000} C_DIS
LIN {X -153.757,Y 245.884,Z 126.492,A -57.981,B 90.000,C 0.000} C_DIS
LIN {X -154.500,Y 245.417,Z 128.832,A -57.808,B 90.000,C 0.000} C_DIS
LIN {X -155.266,Y 244.934,Z 131.075,A -57.629,B 90.000,C 0.000} C_DIS
LIN {X -154.195,Y 243.245,Z 131.075,A -57.629,B 90.000,C 0.000} C_DIS
WAIT SEC 0.1
RET=EKI_SetBool("oxy","torchState",FALSE)
RET = EKI_Send("oxy","torchState")
LIN {X -144.558,Y 228.042,Z 131.075,A -57.629,B 90.000,C 0.000} C_DIS
LIN {X -149.978,Y 224.514,Z 144.399,A -56.257,B 90.000,C 0.000} C_DIS
LIN {X -159.976,Y 239.482,Z 144.399,A -56.257,B 90.000,C 0.000} C_DIS
LIN {X -161.087,Y 241.145,Z 144.399,A -56.257,B 90.000,C 0.000} C_DIS
WAIT SEC 1.75
RET=EKI_SetBool("oxy","torchState",TRUE)
RET = EKI_Send("oxy","torchState")
LIN {X -162.286,Y 240.340,Z 146.440,A -55.971,B 90.000,C 0.000} C_DIS
LIN {X -163.556,Y 239.477,Z 148.412,A -55.668,B 90.000,C 0.000} C_DIS
LIN {X -164.893,Y 238.559,Z 150.315,A -55.348,B 90.000,C 0.000} C_DIS
LIN {X -166.294,Y 237.584,Z 152.141,A -55.010,B 90.000,C 0.000} C_DIS
LIN {X -167.751,Y 236.557,Z 153.893,A -54.658,B 90.000,C 0.000} C_DIS
LIN {X -169.262,Y 235.479,Z 155.568,A -54.292,B 90.000,C 0.000} C_DIS
LIN {X -170.820,Y 234.351,Z 157.163,A -53.911,B 90.000,C 0.000} C_DIS
LIN {X -172.422,Y 233.175,Z 158.681,A -53.519,B 90.000,C 0.000} C_DIS
LIN {X -174.062,Y 231.953,Z 160.117,A -53.115,B 90.000,C 0.000} C_DIS
LIN {X -175.736,Y 230.687,Z 161.475,A -52.700,B 90.000,C 0.000} C_DIS
LIN {X -177.441,Y 229.378,Z 162.751,A -52.275,B 90.000,C 0.000} C_DIS
LIN {X -179.172,Y 228.029,Z 163.947,A -51.842,B 90.000,C 0.000} C_DIS
LIN {X -180.926,Y 226.640,Z 165.064,A -51.400,B 90.000,C 0.000} C_DIS
LIN {X -182.699,Y 225.213,Z 166.097,A -50.950,B 90.000,C 0.000} C_DIS
LIN {X -184.487,Y 223.750,Z 167.050,A -50.494,B 90.000,C 0.000} C_DIS
LIN {X -186.289,Y 222.253,Z 167.924,A -50.031,B 90.000,C 0.000} C_DIS
LIN {X -188.100,Y 220.722,Z 168.714,A -49.562,B 90.000,C 0.000} C_DIS
LIN {X -189.918,Y 219.160,Z 169.423,A -49.089,B 90.000,C 0.000} C_DIS
LIN {X -191.740,Y 217.568,Z 170.052,A -48.611,B 90.000,C 0.000} C_DIS
LIN {X -193.563,Y 215.947,Z 170.596,A -48.129,B 90.000,C 0.000} C_DIS
LIN {X -195.135,Y 214.528,Z 171.000,A -47.710,B 90.000,C 0.000} C_DIS
LIN {X -193.789,Y 213.049,Z 171.000,A -47.710,B 90.000,C 0.000} C_DIS
WAIT SEC 0.1
RET=EKI_SetBool("oxy","torchState",FALSE)
RET = EKI_Send("oxy","torchState")
LIN {X -181.677,Y 199.733,Z 171.000,A -47.710,B 90.000,C 0.000} C_DIS
LIN {X -170.425,Y 209.417,Z 181.693,A -50.861,B 90.000,C 0.000} C_DIS
LIN {X -181.787,Y 223.378,Z 181.693,A -50.861,B 90.000,C 0.000} C_DIS
LIN {X -183.049,Y 224.929,Z 181.693,A -50.861,B 90.000,C 0.000} C_DIS
WAIT SEC 1.75
RET=EKI_SetBool("oxy","torchState",TRUE)
RET = EKI_Send("oxy","torchState")
LIN {X -181.166,Y 226.448,Z 181.062,A -51.339,B 90.000,C 0.000} C_DIS
LIN {X -179.289,Y 227.937,Z 180.350,A -51.812,B 90.000,C 0.000} C_DIS
LIN {X -177.419,Y 229.396,Z 179.562,A -52.281,B 90.000,C 0.000} C_DIS
LIN {X -175.555,Y 230.825,Z 178.705,A -52.745,B 90.000,C 0.000} C_DIS
LIN {X -173.700,Y 232.224,Z 177.785,A -53.204,B 90.000,C 0.000} C_DIS
LIN {X -171.851,Y 233.596,Z 176.809,A -53.659,B 90.000,C 0.000} C_DIS
LIN {X -170.010,Y 234.939,Z 175.783,A -54.109,B 90.000,C 0.000} C_DIS
LIN {X -168.176,Y 236.255,Z 174.710,A -54.555,B 90.000,C 0.000} C_DIS
LIN {X -166.346,Y 237.547,Z 173.600,A -54.998,B 90.000,C 0.000} C_DIS
LIN {X -164.520,Y 238.815,Z 172.456,A -55.437,B 90.000,C 0.000} C_DIS
LIN {X -162.697,Y 240.061,Z 171.285,A -55.873,B 90.000,C 0.000} C_DIS
LIN {X -161.803,Y 240.665,Z 170.701,A -56.086,B 90.000,C 0.000} C_DIS
LIN {X -160.687,Y 239.006,Z 170.701,A -56.086,B 90.000,C 0.000} C_DIS
WAIT SEC 0.1
RET=EKI_SetBool("oxy","torchState",FALSE)
RET = EKI_Send("oxy","torchState")
LIN {X -150.644,Y 224.068,Z 170.701,A -56.086,B 90.000,C 0.000} C_DIS
LIN {X -127.136,Y 238.194,Z 154.999,A -61.909,B 90.000,C 0.000} C_DIS
LIN {X -135.611,Y 254.074,Z 154.999,A -61.909,B 90.000,C 0.000} C_DIS
LIN {X -136.553,Y 255.838,Z 154.999,A -61.909,B 90.000,C 0.000} C_DIS
WAIT SEC 1.75
RET=EKI_SetBool("oxy","torchState",TRUE)
RET = EKI_Send("oxy","torchState")
LIN {X -134.517,Y 256.915,Z 154.027,A -62.364,B 90.000,C 0.000} C_DIS
LIN {X -132.453,Y 257.984,Z 153.108,A -62.823,B 90.000,C 0.000} C_DIS
LIN {X -130.363,Y 259.047,Z 152.241,A -63.287,B 90.000,C 0.000} C_DIS
LIN {X -128.248,Y 260.100,Z 151.426,A -63.753,B 90.000,C 0.000} C_DIS
LIN {X -126.109,Y 261.144,Z 150.662,A -64.224,B 90.000,C 0.000} C_DIS
LIN {X -123.947,Y 262.177,Z 149.950,A -64.697,B 90.000,C 0.000} C_DIS
LIN {X -121.764,Y 263.199,Z 149.288,A -65.173,B 90.000,C 0.000} C_DIS
LIN {X -119.559,Y 264.207,Z 148.679,A -65.652,B 90.000,C 0.000} C_DIS
LIN {X -117.335,Y 265.202,Z 148.121,A -66.134,B 90.000,C 0.000} C_DIS
LIN {X -115.693,Y 265.923,Z 147.742,A -66.488,B 90.000,C 0.000} C_DIS
LIN {X -114.895,Y 264.089,Z 147.742,A -66.488,B 90.000,C 0.000} C_DIS
WAIT SEC 0.1
RET=EKI_SetBool("oxy","torchState",FALSE)
RET = EKI_Send("oxy","torchState")
LIN {X -107.714,Y 247.584,Z 147.742,A -66.488,B 90.000,C 0.000} C_DIS
LIN {X -80.041,Y 257.863,Z 207.593,A -72.756,B 90.000,C 0.000} C_DIS
LIN {X -85.377,Y 275.054,Z 207.593,A -72.756,B 90.000,C 0.000} C_DIS
LIN {X -85.970,Y 276.964,Z 207.593,A -72.756,B 90.000,C 0.000} C_DIS
WAIT SEC 1.75
RET=EKI_SetBool("oxy","torchState",TRUE)
RET = EKI_Send("oxy","torchState")
LIN {X -83.599,Y 277.688,Z 207.911,A -73.245,B 90.000,C 0.000} C_DIS
LIN {X -81.225,Y 278.391,Z 208.256,A -73.735,B 90.000,C 0.000} C_DIS
LIN {X -78.849,Y 279.074,Z 208.627,A -74.223,B 90.000,C 0.000} C_DIS
LIN {X -76.471,Y 279.735,Z 209.025,A -74.711,B 90.000,C 0.000} C_DIS
LIN {X -74.092,Y 280.374,Z 209.450,A -75.197,B 90.000,C 0.000} C_DIS
LIN {X -71.712,Y 280.992,Z 209.898,A -75.683,B 90.000,C 0.000} C_DIS
LIN {X -69.331,Y 281.589,Z 210.370,A -76.168,B 90.000,C 0.000} C_DIS
LIN {X -66.949,Y 282.166,Z 210.863,A -76.652,B 90.000,C 0.000} C_DIS
LIN {X -64.567,Y 282.720,Z 211.380,A -77.136,B 90.000,C 0.000} C_DIS
LIN {X -62.185,Y 283.253,Z 211.918,A -77.618,B 90.000,C 0.000} C_DIS
LIN {X -59.802,Y 283.765,Z 212.476,A -78.099,B 90.000,C 0.000} C_DIS
LIN {X -57.420,Y 284.256,Z 213.053,A -78.580,B 90.000,C 0.000} C_DIS
LIN {X -55.038,Y 284.727,Z 213.647,A -79.060,B 90.000,C 0.000} C_DIS
LIN {X -52.657,Y 285.177,Z 214.259,A -79.538,B 90.000,C 0.000} C_DIS
LIN {X -50.276,Y 285.606,Z 214.887,A -80.016,B 90.000,C 0.000} C_DIS
LIN {X -47.895,Y 286.015,Z 215.531,A -80.494,B 90.000,C 0.000} C_DIS
LIN {X -45.515,Y 286.403,Z 216.189,A -80.970,B 90.000,C 0.000} C_DIS
LIN {X -43.136,Y 286.771,Z 216.861,A -81.446,B 90.000,C 0.000} C_DIS
LIN {X -40.757,Y 287.120,Z 217.545,A -81.921,B 90.000,C 0.000} C_DIS
LIN {X -38.379,Y 287.449,Z 218.241,A -82.395,B 90.000,C 0.000} C_DIS
LIN {X -36.001,Y 287.755,Z 218.950,A -82.869,B 90.000,C 0.000} C_DIS
LIN {X -33.624,Y 288.040,Z 219.669,A -83.342,B 90.000,C 0.000} C_DIS
LIN {X -31.248,Y 288.307,Z 220.397,A -83.814,B 90.000,C 0.000} C_DIS
LIN {X -28.871,Y 288.557,Z 221.132,A -84.286,B 90.000,C 0.000} C_DIS
LIN {X -26.496,Y 288.783,Z 221.876,A -84.758,B 90.000,C 0.000} C_DIS
LIN {X -25.568,Y 288.871,Z 222.167,A -84.942,B 90.000,C 0.000} C_DIS
LIN {X -25.392,Y 286.878,Z 222.167,A -84.942,B 90.000,C 0.000} C_DIS
WAIT SEC 0.1
RET=EKI_SetBool("oxy","torchState",FALSE)
RET = EKI_Send("oxy","torchState")
LIN {X -23.805,Y 268.949,Z 222.167,A -84.942,B 90.000,C 0.000} C_DIS
LIN {X -21.397,Y 269.151,Z 197.078,A -85.455,B 90.000,C 0.000} C_DIS
LIN {X -22.823,Y 287.094,Z 197.078,A -85.455,B 90.000,C 0.000} C_DIS
LIN {X -22.982,Y 289.088,Z 197.078,A -85.455,B 90.000,C 0.000} C_DIS
WAIT SEC 1.75
RET=EKI_SetBool("oxy","torchState",TRUE)
RET = EKI_Send("oxy","torchState")
LIN {X -20.553,Y 289.270,Z 197.641,A -85.936,B 90.000,C 0.000} C_DIS
LIN {X -18.110,Y 289.433,Z 198.143,A -86.420,B 90.000,C 0.000} C_DIS
LIN {X -15.653,Y 289.577,Z 198.583,A -86.906,B 90.000,C 0.000} C_DIS
LIN {X -13.185,Y 289.699,Z 198.960,A -87.394,B 90.000,C 0.000} C_DIS
LIN {X -10.707,Y 289.802,Z 199.274,A -87.884,B 90.000,C 0.000} C_DIS
LIN {X -8.221,Y 289.883,Z 199.524,A -88.375,B 90.000,C 0.000} C_DIS
LIN {X -6.413,Y 289.929,Z 199.668,A -88.733,B 90.000,C 0.000} C_DIS
LIN {X -6.369,Y 287.930,Z 199.668,A -88.733,B 90.000,C 0.000} C_DIS
WAIT SEC 0.1
RET=EKI_SetBool("oxy","torchState",FALSE)
RET = EKI_Send("oxy","torchState")
LIN {X -5.971,Y 269.934,Z 199.668,A -88.733,B 90.000,C 0.000} C_DIS
LIN {X -4.062,Y 269.969,Z 195.603,A -89.138,B 90.000,C 0.000} C_DIS
LIN {X -4.333,Y 287.967,Z 195.603,A -89.138,B 90.000,C 0.000} C_DIS
LIN {X -4.363,Y 289.967,Z 195.603,A -89.138,B 90.000,C 0.000} C_DIS
WAIT SEC 1.75
RET=EKI_SetBool("oxy","torchState",TRUE)
RET = EKI_Send("oxy","torchState")
LIN {X -2.024,Y 289.991,Z 196.484,A -89.600,B 90.000,C 0.000} C_DIS
LIN {X 0.319,Y 289.999,Z 197.357,A -90.063,B 90.000,C 0.000} C_DIS
LIN {X 2.665,Y 289.985,Z 198.219,A -90.527,B 90.000,C 0.000} C_DIS
LIN {X 5.015,Y 289.953,Z 199.071,A -90.991,B 90.000,C 0.000} C_DIS
LIN {X 7.367,Y 289.903,Z 199.914,A -91.456,B 90.000,C 0.000} C_DIS
LIN {X 9.723,Y 289.835,Z 200.748,A -91.921,B 90.000,C 0.000} C_DIS
LIN {X 12.081,Y 289.748,Z 201.573,A -92.388,B 90.000,C 0.000} C_DIS
LIN {X 14.443,Y 289.638,Z 202.385,A -92.855,B 90.000,C 0.000} C_DIS
LIN {X 16.806,Y 289.509,Z 203.188,A -93.322,B 90.000,C 0.000} C_DIS
LIN {X 19.172,Y 289.362,Z 203.982,A -93.791,B 90.000,C 0.000} C_DIS
LIN {X 21.540,Y 289.197,Z 204.767,A -94.260,B 90.000,C 0.000} C_DIS
LIN {X 23.909,Y 289.013,Z 205.543,A -94.729,B 90.000,C 0.000} C_DIS
LIN {X 26.280,Y 288.805,Z 206.306,A -95.199,B 90.000,C 0.000} C_DIS
LIN {X 28.652,Y 288.578,Z 207.060,A -95.670,B 90.000,C 0.000} C_DIS
LIN {X 29.762,Y 288.469,Z 207.411,A -95.891,B 90.000,C 0.000} C_DIS
LIN {X 29.557,Y 286.479,Z 207.411,A -95.891,B 90.000,C 0.000} C_DIS
WAIT SEC 0.1
RET=EKI_SetBool("oxy","torchState",FALSE)
RET = EKI_Send("oxy","torchState")
LIN {X 27.710,Y 268.574,Z 207.411,A -95.891,B 90.000,C 0.000} C_DIS
LIN {X 24.186,Y 268.915,Z 179.974,A -95.139,B 90.000,C 0.000} C_DIS
LIN {X 25.798,Y 286.842,Z 179.974,A -95.139,B 90.000,C 0.000} C_DIS
LIN {X 25.977,Y 288.834,Z 179.974,A -95.139,B 90.000,C 0.000} C_DIS
WAIT SEC 1.75
RET=EKI_SetBool("oxy","torchState",TRUE)
RET = EKI_Send("oxy","torchState")
LIN {X 23.678,Y 289.032,Z 179.013,A -94.683,B 90.000,C 0.000} C_DIS
LIN {X 21.403,Y 289.209,Z 177.992,A -94.232,B 90.000,C 0.000} C_DIS
LIN {X 19.154,Y 289.367,Z 176.913,A -93.787,B 90.000,C 0.000} C_DIS
LIN {X 16.932,Y 289.505,Z 175.775,A -93.347,B 90.000,C 0.000} C_DIS
LIN {X 14.740,Y 289.625,Z 174.580,A -92.913,B 90.000,C 0.000} C_DIS
LIN {X 12.578,Y 289.727,Z 173.329,A -92.486,B 90.000,C 0.000} C_DIS
LIN {X 10.449,Y 289.812,Z 172.023,A -92.065,B 90.000,C 0.000} C_DIS
LIN {X 8.353,Y 289.880,Z 170.662,A -91.651,B 90.000,C 0.000} C_DIS
LIN {X 6.293,Y 289.932,Z 169.247,A -91.243,B 90.000,C 0.000} C_DIS
LIN {X 4.270,Y 289.968,Z 167.780,A -90.844,B 90.000,C 0.000} C_DIS
LIN {X 2.285,Y 289.991,Z 166.260,A -90.451,B 90.000,C 0.000} C_DIS
LIN {X 0.340,Y 290.000,Z 164.690,A -90.067,B 90.000,C 0.000} C_DIS
LIN {X -0.215,Y 290.000,Z 164.227,A -89.957,B 90.000,C 0.000} C_DIS
LIN {X -0.214,Y 288.000,Z 164.227,A -89.957,B 90.000,C 0.000} C_DIS
WAIT SEC 0.1
RET=EKI_SetBool("oxy","torchState",FALSE)
RET = EKI_Send("oxy","torchState")
LIN {X -0.200,Y 270.000,Z 164.227,A -89.957,B 90.000,C 0.000} C_DIS
LIN {X 49.853,Y 265.358,Z 160.640,A -100.640,B 90.000,C 0.000} C_DIS
LIN {X 53.177,Y 283.048,Z 160.640,A -100.640,B 90.000,C 0.000} C_DIS
LIN {X 53.546,Y 285.014,Z 160.640,A -100.640,B 90.000,C 0.000} C_DIS
WAIT SEC 1.75
RET=EKI_SetBool("oxy","torchState",TRUE)
RET = EKI_Send("oxy","torchState")
LIN {X 55.837,Y 284.572,Z 161.535,A -101.101,B 90.000,C 0.000} C_DIS
LIN {X 58.130,Y 284.113,Z 162.421,A -101.563,B 90.000,C 0.000} C_DIS
LIN {X 60.421,Y 283.635,Z 163.297,A -102.026,B 90.000,C 0.000} C_DIS
LIN {X 62.712,Y 283.138,Z 164.166,A -102.489,B 90.000,C 0.000} C_DIS
LIN {X 64.999,Y 282.617,Z 165.028,A -102.952,B 90.000,C 0.000} C_DIS
LIN {X 67.284,Y 282.080,Z 165.888,A -103.416,B 90.000,C 0.000} C_DIS
LIN {X 69.566,Y 281.526,Z 166.745,A -103.880,B 90.000,C 0.000} C_DIS
LIN {X 71.843,Y 280.952,Z 167.602,A -104.344,B 90.000,C 0.000} C_DIS
LIN {X 74.116,Y 280.362,Z 168.459,A -104.808,B 90.000,C 0.000} C_DIS
LIN {X 76.383,Y 279.755,Z 169.320,A -105.272,B 90.000,C 0.000} C_DIS
LIN {X 78.645,Y 279.132,Z 170.183,A -105.735,B 90.000,C 0.000} C_DIS
LIN {X 80.896,Y 278.485,Z 171.055,A -106.198,B 90.000,C 0.000} C_DIS
LIN {X 83.141,Y 277.823,Z 171.934,A -106.660,B 90.000,C 0.000} C_DIS
LIN {X 85.377,Y 277.145,Z 172.823,A -107.122,B 90.000,C 0.000} C_DIS
LIN {X 87.603,Y 276.450,Z 173.722,A -107.583,B 90.000,C 0.000} C_DIS
LIN {X 89.819,Y 275.738,Z 174.635,A -108.042,B 90.000,C 0.000} C_DIS
LIN {X 92.023,Y 275.010,Z 175.563,A -108.501,B 90.000,C 0.000} C_DIS
LIN {X 94.215,Y 274.267,Z 176.506,A -108.958,B 90.000,C 0.000} C_DIS
LIN {X 96.394,Y 273.509,Z 177.468,A -109.414,B 90.000,C 0.000} C_DIS
LIN {X 97.064,Y 273.274,Z 177.766,A -109.555,B 90.000,C 0.000} C_DIS
LIN {X 96.395,Y 271.389,Z 177.766,A -109.555,B 90.000,C 0.000} C_DIS
WAIT SEC 0.1
RET=EKI_SetBool("oxy","torchState",FALSE)
RET = EKI_Send("oxy","torchState")
LIN {X 90.370,Y 254.427,Z 177.766,A -109.555,B 90.000,C 0.000} C_DIS
LIN {X 66.621,Y 261.652,Z 194.663,A -104.285,B 90.000,C 0.000} C_DIS
LIN {X 71.063,Y 279.095,Z 194.663,A -104.285,B 90.000,C 0.000} C_DIS
LIN {X 71.556,Y 281.033,Z 194.663,A -104.285,B 90.000,C 0.000} C_DIS
WAIT SEC 1.75
RET=EKI_SetBool("oxy","torchState",TRUE)
RET = EKI_Send("oxy","torchState")
LIN {X 73.762,Y 280.462,Z 195.691,A -104.735,B 90.000,C 0.000} C_DIS
LIN {X 75.945,Y 279.879,Z 196.761,A -105.182,B 90.000,C 0.000} C_DIS
LIN {X 78.113,Y 279.279,Z 197.850,A -105.626,B 90.000,C 0.000} C_DIS
LIN {X 80.279,Y 278.666,Z 198.938,A -106.071,B 90.000,C 0.000} C_DIS
LIN {X 82.450,Y 278.032,Z 200.001,A -106.518,B 90.000,C 0.000} C_DIS
LIN {X 84.636,Y 277.374,Z 201.019,A -106.969,B 90.000,C 0.000} C_DIS
LIN {X 86.839,Y 276.693,Z 201.985,A -107.424,B 90.000,C 0.000} C_DIS
